	r_ApparentPower					: REAL;
	r_ActivePower					: REAL;
	r_ReactivePower					: REAL;
	r_ACVoltageD7					: REAL;
	r_VoltageDroop					: REAL;
	r_ACVoltageSupply				: REAL;
	r_FrequencyD7					: REAL;
	r_FrequencyDroop				: REAL;
	r_FrequencySupply				: REAL;
	r_CurrentUnbalance				: REAL;
	r_DCPower						: REAL;
	r_DCVoltage						: REAL;
	r_DCCurrent						: REAL;
	r_ACCurrent						: REAL;
	r_ActiveCurrent					: REAL;
	r_ReactiveCurrent				: REAL;
	r_LoadPercent					: REAL; //%
	r_D7SyncError					: REAL;
	r_Pmin							: REAL;
	r_Pmax							: REAL;
	r_QMax							: REAL;
	r_Qmin							: REAL;
	r_Pset							: REAL;
	r_Qset							: REAL;
	r_ACcurrentLimit				: REAL; 
	r_OverCurrentValue				: REAL; // overcurrent ratio 0 .. 1.25 x rated current
	r_ModulationIndex				: REAL;
	
	r_TemperatureInverter			: REAL;
	r_TemperatureGridChoke			: ARRAY [1..3] OF REAL;
	r_TemperatureCMChoke			: ARRAY [1..4] OF REAL;
	r_TemperatureMax				: REAL;
	AddTemperatures					: ST_Inverter_additionalTemperatures;
	w_TemperatureFaultWord			: WORD;
	w_OperationHours				: WORD;
	
	e_PowerMode						: ePowerModes;
	e_InverterMode					: eInverterModes;
	e_Status						: eStatusPowermodule;
	e_ThrottlingStatus					: ePowerModuleThrottlingState;		
	ui_InverterCommStatus			: UINT;
	ui_BuscouplerCommStatus			: UINT;
	
	b_MccbTripOK					: BOOL;
	b_MccbUvr24VdcOK				: BOOL;
	b_MccbFb						: BOOL;
	b_FanFb							: BOOL;
	b_DCcontactorFb					: BOOL;
	b_PrechargeContactor			: BOOL;
	b_LimiterActive					: BOOL;
	
	
	StatusWord						: ST_Inverter_StatusWord;
	UgridStatusWord					: ST_Inverter_UgridStatusWord;
	GridcodeStatusWord				: ST_Inverter_LineState;
	Events							: ST_Powermodule_Events;
	controldata						: ST_Inverter_write;
	
END_STRUCT
END_TYPE

// ---- POUs/Objects/PowerStack/_Structs/ST_PowerModule_set.TcDUT
TYPE ST_PowerModule_set :
STRUCT
	//commands
	r_ActivePower					: REAL;
	r_ReactivePower					: REAL;
	r_NomFrequency					: REAL;
	r_NomVoltage					: REAL;
	r_FrequencyDroop				: REAL;
	r_VoltageDroop					: REAL;
	r_Pmax							: REAL;
	r_Pmin							: REAL;
	r_ACcurrentLimit				: REAL;
	i_PowerChangeRate				: INT; // % nominal power / s
	r_overcurrentFactor				: REAL;
	r_DroopMinimum					: REAL := 0.1;
	r_DroopIslandMode				: REAL := 0.1;
	r_DroopMaximum					: REAL := 10; //%
	
	//WRITE DATA Buscoupler
	b_FanContactor					: BOOL;
	b_D7SyncRequest					: BOOL;
	b_QuickstopInactive				: BOOL;
	b_gridcodeEnable				: BOOL;
	b_ExtgridCodeTrip				: BOOL;
END_STRUCT
END_TYPE

// ---- POUs/Objects/PowerStack/_Structs/ST_Powerstack_Calibration.TcDUT
TYPE ST_Powerstack_Calibration:
STRUCT
	Master				: ST_PowerModule_calibration;
	Slave				: ST_PowerModule_calibration;
END_STRUCT
END_TYPE

// ---- POUs/Objects/PowerStack/_Structs/ST_PowerStack_get.TcDUT
TYPE ST_PowerStack_get :
STRUCT
	// ENUMS
	e_State							: eStatusPowerStack;
	e_PowerState					: ePowerstate;
	e_InverterMode					: eInverterModes;			//0=AFE, Micro, Island, transition
	e_PowerMode						: ePowerModes;				//0=IsoChronous, 1= Droop
	e_ThrottlingStatus				: ePowerModuleThrottlingState;
	
	//POWER DATA (REALS)
	r_VoltageDroop					: REAL;				
	r_FrequencyDroop				: REAL;
	r_ACVoltageD7					: REAL; 
	r_FrequencyD7					: REAL; 
	r_ActivePower					: REAL;
	r_ReactivePower					: REAL;
	r_Pmin							: REAL;
	r_Pmax							: REAL; 
	r_QMax							: REAL;
	r_QMin							: REAL;	
	r_Smax							: REAL;
	r_ACcurrentLimit				: REAL;
	r_ACcurrentLimitMax				: REAL;
	r_PowerChangeRate				: REAL;
	r_ApparentPower					: REAL;
	r_CosPhi						: REAL;
	r_AcCurrent						: REAL;
	r_DCPower						: REAL;
	r_DCVoltage						: REAL;
	r_DCcurrent						: REAL;
	r_ACVoltageSupply				: REAL;
	r_FrequencySupply				: REAL;
	r_LoadPercent					: REAL; //%
	r_RatedCurrent					: REAL;
	r_RatedPower					: REAL;
	r_OvercurrentValueAct			: REAL; //actual overcurrent value
	r_OvercurrentValueMax			: REAL; //max overcurrent value
	r_ThrottlingValueAct			: REAL; // %percentage , inverse of overcurrent with 100%
	
	//Booleans
	b_GridTied						: BOOL;
	b_GridCodeCheckActive			: BOOL;
	b_GridCodeOK					: BOOL := TRUE;
	b_GridACdetected				: BOOL;
	b_InverterGridFormingMode		: BOOL;
	b_ACDetected					: BOOL;
	b_DCDetected					: BOOL;
	b_InverterRunning				: BOOL;
	b_StartedState					: BOOL;
	b_ControlEnabled				: BOOL;
	b_EcomodeAvailable				: BOOL;
	b_StartEnabled					: BOOL;				

	//Temperatures
	r_MaxTemperature				: REAL;
	
	//timers
	t_ShiftHoldTimeRemaining		: TIME;
	t_GridCodeReconnectTime			: TIME;
	//structs
	Events							: ST_PowerStack_Events;
	
	//Sublevel data
	PowermoduleMaster				: REFERENCE TO ST_PowerModule_get();
	PowermoduleSlave				: REFERENCE TO ST_PowerModule_get();
	Netcontactor					: REFERENCE TO ST_Netcontactor_get();
	
END_STRUCT
END_TYPE

// ---- POUs/Objects/PowerStack/_Structs/ST_Powerstack_LOMParams.TcDUT
TYPE ST_Powerstack_LOMParams :
STRUCT
	ForceSlowDetection	: BOOL := FALSE;
	FreqFilterLength	: UINT := 5; // samples 
	DetectionTimeFast_ms: UINT := 50; // milliseconds
	DetectionTimeSlow_ms: UINT := 1000; // milliseconds
	RoCofLimit			: REAL := 0.5; // Hz/s
	PowerPulseSize		: REAL := 0.5; // %, of rated power during ugrid to enable LOM detection.
	EnablePowerPulse	: BOOL := TRUE;
END_STRUCT
END_TYPE

// ---- POUs/Objects/PowerStack/_Structs/ST_PowerStack_params.TcDUT
TYPE ST_PowerStack_params :
STRUCT
	b_SoftStartEnable		: BOOL := TRUE;
	b_StandbyEnable			: BOOL := TRUE;
	b_GridcodesEnabled		: BOOL := TRUE;
	r_DroopMinimum			: REAL := 0.0;
	r_DroopIslandMode		: REAL := 0.1;
	r_DroopMaximum			: REAL := 10; //%
	r_ReactiveOffset		: REAL := 0;
	ui_DeratingStack		: UINT := 5; // %
	ui_DeratingLimCooling	: UINT := 80; // %
	i_MaxPowerChangeRate	: INT := 500; // %/s
	ui_OvercurrentRating	: UINT := 150; // %
	i_ChargeOnlyIdlePower	: INT := -3;
	r_ActiveSetpointGain	: REAL := 1; 
	r_ReactiveSetpointGain  : REAL := 1;
	
	//AC drive limits
	r_FreqLowLimit			: REAL := 48;
	r_FreqHighLimit			: REAL := 52; 
	ui_FreqLimitTripDelay	: UINT := 2000; // milliseconds
	FreqVoltageShift		: st_powerstack_ShiftingParams;
	
	PowermoduleMaster		: ST_PowerModule_params;
	PowermoduleSlave		: ST_PowerModule_params;
	LOM						: ST_Powerstack_LOMParams;
END_STRUCT
END_TYPE

// ---- POUs/Objects/PowerStack/_Structs/ST_PowerStack_Set.TcDUT
TYPE ST_PowerStack_Set :
STRUCT
	//WRITE
	b_NetcontactorHoldClose			: BOOL; // used when input breaker or external PSB breaker must be controlled instead of netcontactor.
	b_ExtGridConnected				: BOOL;
	b_DisableShifting				: BOOL;
	b_slowLom						: BOOL;
	b_automaticswitching			: BOOL;
	b_GridCodeEnable				: BOOL := TRUE;
	e_InverterMode					: eInverterModes;			//0=AFE, 1= ugrid, 2, island
	e_PowerMode						: ePowerModes;				//
	e_NetconClosingRequest			: eNetcontMode;
	e_PowerLimitingMode				: ePLM;
	r_VoltageDroop					: REAL;				
	r_FrequencyDroop				: REAL;
	r_NominalOutputVoltage			: REAL := 400; //R/W
	r_NominalOutputFrequency		: REAL := 50; //R/W
	r_ActivePower					: REAL; //R/W
	r_ReactivePower					: REAL; //R/W
	
	//limits
	r_Pmax							: REAL;
	r_Pmin							: REAL;
	r_ACcurrentLimit				: REAL;
	
END_STRUCT
END_TYPE

// ---- POUs/Objects/ProtectionSystems/FireDetection/_Enums/eCOAlarmStatus.TcDUT
{attribute 'qualified_only'}
{attribute 'strict'}
{attribute 'tostring'}
TYPE eCOAlarmStatus :
(
	Error			:= 0,
	Normal 			:= 1,
	WarningLevel1 	:= 2,
	WarningLevel2 	:= 3,
	Alarm 			:= 4
);
END_TYPE

// ---- POUs/Objects/ProtectionSystems/FireDetection/_Enums/eSmokeDetectAlarmStatus.TcDUT
{attribute 'qualified_only'}
{attribute 'strict'}
{attribute 'tostring'}
TYPE eSmokeDetectAlarmStatus :
(
	Error := 0,
	Normal := 1,
	Alarm := 2
);
END_TYPE

// ---- POUs/Objects/ProtectionSystems/FireDetection/_Structs/ST_CODetectors.TcDUT
TYPE ST_CODetectors :
STRUCT
	State 			: 	eCOAlarmStatus;
	b_CoValuesOK	: 	BOOL;
	Value 			:  	ARRAY[0..3] OF REAL;	//-1 if inoperative. [0]=mean [1]=CO1 [2]=CO2 [3]=max
END_STRUCT
END_TYPE

// ---- POUs/Objects/ProtectionSystems/FireDetection/_Structs/ST_FireDetection_get.TcDUT
TYPE ST_FireDetection_get :
STRUCT
	b_FireAlarm		: 	BOOL;
	SmokeDetectors 	:	ST_SmokeDetectors;
	CODetectors		:	ST_CODetectors;
	Events			:	ST_FireSystem_Events;
END_STRUCT
END_TYPE

// ---- POUs/Objects/ProtectionSystems/FireDetection/_Structs/st_Firedetection_params.TcDUT
TYPE st_Firedetection_params :
STRUCT
	r_COwarningLevel_1				: REAL := 10;
	r_COwarningLevel_2				: REAL := 20;
	r_COalarmLevel					: REAL := 120;
	r_COrange						: REAL := 500;
END_STRUCT
END_TYPE

// ---- POUs/Objects/ProtectionSystems/FireDetection/_Structs/ST_FireDetection_set.TcDUT
TYPE ST_FireDetection_set :
STRUCT
	SilenceSounder	:	BOOL; //only disables currently activated alarm.
	TestSounder		:	BOOL;
END_STRUCT
END_TYPE

// ---- POUs/Objects/ProtectionSystems/FireDetection/_Structs/ST_FireSystem_Events.TcDUT
TYPE ST_FireSystem_Events :
STRUCT
	CODetFault		:	BOOL;
	CODetWarning1	:	BOOL;
	CODetWarning2	: 	BOOL;
	CODetAlarm		:	BOOL;
	SmokeDetFault	:	BOOL;
	SmokeDetAlarm	:	BOOL;
	AlarmMuted		:	BOOL;
END_STRUCT
END_TYPE

// ---- POUs/Objects/ProtectionSystems/FireDetection/_Structs/ST_SmokeDetectors.TcDUT
TYPE ST_SmokeDetectors :
STRUCT
	State : eSmokeDetectAlarmStatus;
END_STRUCT
END_TYPE

// ---- POUs/Objects/ProtectionSystems/FireDetection/_Structs/ST_SmokeDetIO.TcDUT
TYPE ST_SmokeDetIO :
STRUCT
	Signal_OK 	: BOOL;
	Power_OK 	: BOOL;
END_STRUCT
END_TYPE

// ---- POUs/Objects/ProtectionSystems/InsulationMonitoring/_Structs/ST_InsulationMonitor_get.TcDUT
TYPE ST_InsulationMonitor_get :
STRUCT
	b_Enabled							: BOOL;	
	b_PENlinkDetected					: BOOL;
	b_Warning							: BOOL;
	e_EarthingSystemDetected			: eEarthingSystems;
	b_PENlinkOperatedFault				: BOOL;
	b_EarthingSystemMismatch			: BOOL;
	b_NoEarthingSystemSet				: BOOL;
END_STRUCT
END_TYPE

// ---- POUs/Objects/ProtectionSystems/InsulationMonitoring/_Structs/ST_InsulationMonitor_params.TcDUT
TYPE ST_InsulationMonitor_params :
STRUCT
	i_EarthSystemDetectionDelay		:INT := 60; // Seconds
END_STRUCT
END_TYPE

// ---- POUs/Objects/ProtectionSystems/InsulationMonitoring/_Structs/St_InsulationMonitor_PassThrough.TcDUT
TYPE St_InsulationMonitor_PassThrough :
STRUCT
	b_NetContFB				: BOOL;
	b_MccbfbMaster			: BOOL;
	b_MccbfbSlave			: BOOL;
	b_ACdetected			: BOOL;
	b_PENlinkFB				: BOOL;	
END_STRUCT
END_TYPE

// ---- POUs/Objects/ProtectionSystems/InsulationMonitoring/_Structs/ST_InsulationMonitor_set.TcDUT
TYPE ST_InsulationMonitor_set :
STRUCT
	b_enable			: BOOL;
 	e_EarthingSystem	: eEarthingSystems := eEarthingSystems.TN;
END_STRUCT
END_TYPE

// ---- POUs/Objects/ProtectionSystems/OvercurrentProtection/_Structs/ST_OvercurrentProtection_Events.TcDUT
TYPE ST_OvercurrentProtection_Events :
STRUCT
	Input	:ARRAY [1..2] OF ARRAY [1..4] OF FB_Overcurrentdetect(); //FB_UpperLimitAndTimeExceeded();
	Output	:ARRAY [1..3] OF ARRAY [1..4] OF FB_Overcurrentdetect();
END_STRUCT
END_TYPE

// ---- POUs/Objects/ProtectionSystems/OvercurrentProtection/_Structs/ST_OvercurrentProtection_get.TcDUT
TYPE ST_OvercurrentProtection_get :
STRUCT
	//Overcurrent Powerlocks
	r_TotalOutputCurrentLimit			: REAL := 0;
	r_TotalInputCurrentLimit			: REAL := 0;
	b_OutputWarning						: BOOL;
	b_InputWarning						: BOOL;
	b_OutputAlarm						: BOOL;
	b_InputAlarm						: BOOL;
	r_PeakCurrent						: REAL;
	t_PeakCurrentDuration				: TIME;
	s_locationPeak						: STRING;
	
	Events								: ST_OvercurrentProtection_events;
END_STRUCT
END_TYPE

// ---- POUs/Objects/ProtectionSystems/OvercurrentProtection/_Structs/ST_OvercurrentProtection_InternalLinking.TcDUT
TYPE ST_OvercurrentProtection_InternalLinking :
STRUCT
	a_r_CurrentInput			: ARRAY [1..2] OF ARRAY[1..4] OF REAL; //first array of powerlockset, second of powerlock
	a_r_CurrentOutput			: ARRAY [1..3] OF ARRAY[1..4] OF REAL;
	b_InputSectionAvailable 	: BOOL;
	b_thirdOutputAvailable 		: BOOL;
END_STRUCT
END_TYPE

// ---- POUs/Objects/ProtectionSystems/OvercurrentProtection/_Structs/ST_OvercurrentProtection_Params.TcDUT
TYPE ST_OvercurrentProtection_Params :
STRUCT
	ui_OCPtripTime		: UINT := 900; //Seconds
	ui_Ik				: UINT := 16; // Short circuit capacity of component to be protected [Ik/s]
	ui_Irated			: UINT := 400; // rated current 
	ui_gain				: UINT := 10; //gain for tuning calculated remaining time during overcurrent.
	OutputNormalShutdownDelay : TIME := T#5S;
END_STRUCT
END_TYPE

// ---- POUs/Objects/ProtectionSystems/OvercurrentProtection/_Structs/ST_OvercurrentProtection_set.TcDUT
TYPE ST_OvercurrentProtection_set :
STRUCT
	ui_PowerlockInputCurrentLimit			: ARRAY [1..2] OF UINT := [400,400];
	ui_PowerlockOutputCurrentLimit			: ARRAY [1..3] OF UINT := [400,400,400];
END_STRUCT
END_TYPE

// ---- POUs/Objects/ProtectionSystems/ResidualCurrentMonitoring/_Structs/ST_ResidualCurrentMonitor_get.TcDUT
TYPE ST_ResidualCurrentMonitor_get :
STRUCT
	b_prewarning			: BOOL;
END_STRUCT
END_TYPE

// ---- POUs/Objects/ProtectionSystems/SurgeProtection/_Structs/ST_Surgeprotection_get.TcDUT
TYPE ST_Surgeprotection_get :
STRUCT
	b_Type12_OK				: BOOL;
	b_Type3_OK				: BOOL;			
END_STRUCT
END_TYPE

// ---- POUs/Objects/ProtectionSystems/_Struct/ST_ProtectionSystems_get.TcDUT
TYPE ST_ProtectionSystems_get :
STRUCT
	//Fire Detection System
	FireDetection						: ST_Firedetection_get;
	
	//InsulationMonitor
	Insulation							: ST_InsulationMonitor_get;
	
	//MRCDB
	MRCDB								: ST_ResidualCurrentMonitor_get;
	
	//Surge protection
	Surge								: ST_SurgeProtection_get;
	
	//Overcurrent protection
	OvercurrentProtection				: ST_OverCurrentProtection_Get;
	
END_STRUCT
END_TYPE

// ---- POUs/Objects/ProtectionSystems/_Struct/ST_ProtectionSystems_Params.TcDUT
TYPE ST_ProtectionSystems_Params :
STRUCT
	InsulationMonitor				: ST_InsulationMonitor_params;
	firedetection					: ST_Firedetection_params;
	OCP								: ST_Overcurrentprotection_params;
END_STRUCT
END_TYPE

// ---- POUs/Objects/ProtectionSystems/_Struct/ST_ProtectionSystems_set.TcDUT
TYPE ST_ProtectionSystems_set :
STRUCT
	//Fire Detection System
	FireDetection						: ST_Firedetection_set;
	
	//InsulationMonitor
	Insulation							: ST_InsulationMonitor_set;
	
	//OCP
	OvercurrentProtection				: ST_OvercurrentProtection_set;
END_STRUCT
END_TYPE

// ---- POUs/Objects/PeakshaveBox/DUTs/eWago750495_ACDataID_1.TcDUT
{attribute 'qualified_only'}
{attribute 'strict'}
{attribute 'to_String'}
TYPE eWago750495_ACDataID_1 :
(
	//only RMS and peak values are declared
	//Voltages
	VoltageL1N_RMS			:= 4,
	VoltageL2N_RMS 			:= 5,
	VoltageL3N_RMS			:= 6,
	VoltageL1L2_RMS			:= 31,
	VoltageL2L3_RMS 		:= 32,
	VoltageL3L1_RMS			:= 33,
	VoltageL1N_Peak 		:= 91,
	VoltageL2N_Peak 		:= 92,
	VoltageL3N_Peak 		:= 93,
	
	//Currents
	CurrentL1_RMS			:= 1,
	CurrentL2_RMS			:= 2,
	CurrentL3_RMS			:= 3,
	CurrentN_RMS			:= 97,
	CurrentL1_Peak			:= 94,
	CurrentL2_Peak			:= 95,
	CurrentL3_Peak			:= 96,
	                           
	//Power                    
	ActivePowerL1			:= 07,
	ActivePowerL2			:= 08,
	ActivePowerL3			:= 09,
	ReactivePowerL1			:= 10,
	ReactivePowerL2			:= 11,
	ReactivePowerL3			:= 12,
	ApparentPowerL1			:= 13,
	ApparentPowerL2			:= 14,
	ApparentPowerL3			:= 15,
	
	//Energy
	ActiveEnergyTotal			:= 73,
	ActiveEnergyImport			:= 74,
	ActiveEnergyExport			:= 75,
	ReactiveEnergyTotal			:= 85,
	ReactiveEnergyInductive		:= 86,
	AReactiveEnergyCapacitive	:= 87,
	
	//Frequency
	FrequencyL1				:= 16,
	FrequencyL2				:= 17,
	FrequencyL3				:= 18,
	                           
	//Phase Angle              
	PhaseAngleL1			:= 19,
	PhaseAngleL2			:= 20,
	PhaseAngleL3			:= 21,
	
	//PowerFactor
	PowerFactorL1			:= 25,
	PowerFactorL2			:= 26,
	PowerFactorL3			:= 27
) USINT;
END_TYPE

// ---- POUs/Objects/PeakshaveBox/DUTs/eWago750495_HarmonicsDataID_1.TcDUT
{attribute 'qualified_only'}
{attribute 'strict'}
{attribute 'to_String'}
TYPE eWago750495_HarmonicsDataID_1 :
(
	Current_RMS 		:= 001,
	Voltage_RMS 		:= 002,
	CurrentTHD			:= 003,
	VoltageTHD			:= 004
	
	//harmonics not declared for now
);
END_TYPE

// ---- POUs/Objects/PeakshaveBox/DUTs/eWago750495_MeasureGroupID_1.TcDUT
{attribute 'qualified_only'}
{attribute 'strict'}
{attribute 'to_String'}
TYPE eWago750495_MeasureGroupID_1 :
(
	ac := 10,
	harmonicsL1 := 20,
	harmonicsL2 := 21,
	harmonicsL3	:= 22
) USINT;
END_TYPE

// ---- POUs/Objects/PeakshaveBox/DUTs/eWago750495_StatDataID_1.TcDUT
{attribute 'qualified_only'}
{attribute 'strict'}
TYPE eWago750495_StatDataID_1 :
(
	Phase1 := 0,
	Phase2 := 1,
	Phase3 := 2,
	IOmodule:= 3
)USINT;
END_TYPE

// ---- POUs/Objects/PeakshaveBox/DUTs/ST_Wago750495_Data_1.TcDUT
TYPE ST_Wago750495_Data_1 :
STRUCT
	//Voltages
	r_VoltageL1N_RMS				: REAL;
	r_VoltageL2N_RMS 				: REAL;
	r_VoltageL3N_RMS				: REAL;
	r_VoltageL1L2_RMS				: REAL;
	r_VoltageL2L3_RMS 				: REAL;
	r_VoltageL3L1_RMS				: REAL;
	r_VoltageL1N_Peak 				: REAL;
	r_VoltageL2N_Peak 				: REAL;
	r_VoltageL3N_Peak 				: REAL;
	                            	      
	//Currents                  	      
	r_CurrentL1_RMS					: REAL;
	r_CurrentL2_RMS					: REAL;
	r_CurrentL3_RMS					: REAL;
	r_CurrentN_RMS					: REAL;
	r_CurrentL1_Peak				: REAL;
	r_CurrentL2_Peak				: REAL;
	r_CurrentL3_Peak				: REAL;
	                            	      
	//Power                     	      
	r_ActivePowerL1					: REAL;
	r_ActivePowerL2					: REAL;
	r_ActivePowerL3					: REAL;
	r_ReactivePowerL1				: REAL;
	r_ReactivePowerL2				: REAL;
	r_ReactivePowerL3				: REAL;
	r_ApparentPowerL1				: REAL;
	r_ApparentPowerL2				: REAL;
	r_ApparentPowerL3				: REAL;
	
	//Energy
	r_ActiveEnergyTotal				: REAL;
	r_ActiveEnergyImport			: REAL;
	r_ActiveEnergyExport			: REAL;
	r_ReactiveEnergyTotal			: REAL;
	r_ReactiveEnergyInductive		: REAL;
	r_AReactiveEnergyCapacitive		: REAL;
	
	//Frequency
	r_FrequencyL1					: REAL;
	r_FrequencyL2					: REAL;
	r_FrequencyL3					: REAL;
	                        		      
	//Phase Angle           		      
	r_PhaseAngleL1					: REAL;
	r_PhaseAngleL2					: REAL;
	r_PhaseAngleL3					: REAL;
	                        		      
	//PowerFactor           		      
	r_PowerFactorL1					: REAL;
	r_PowerFactorL2					: REAL;
	r_PowerFactorL3					: REAL;
	
	
END_STRUCT
END_TYPE

// ---- POUs/Objects/PeakshaveBox/DUTs/ST_Wago750495_ExtStatusWord_1.TcDUT
TYPE ST_Wago750495_ExtStatusWord_1 :
STRUCT
	b_IncreasedMeasErr			: BOOL; //Stat 1 query L1,L2,L3:: increase measurement error of selected phase
	b_CurrentClipping			: BOOL; //Stat 2 query L1,L2,L3:: current out of measurable range of selected phase
	b_VoltageClipping			: BOOL; //Stat 3 query L1,L2,L3:: voltage out of measurable range of selected phase
	b_NoZeroCrossings			: BOOL; //Stat 4 query L1,L2,L3:: Zero Crossings missing of selected phase
	b_OverCurrent				: BOOL; //Stat 5 query L1,L2,L3:: Overcurrent of selected phase
	b_OverVoltage				: BOOL; //Stat 6- query L1,L2,L3: OverVoltage of selected phase.
	b_RotaryField				: BOOL; //Stat 6- query IO: 0:Clockwise, 1: counterclockwise
	b_UnderVoltage				: BOOL; //Stat 7- query L1,L2,L3: UnderVoltage of selected phase

END_STRUCT
END_TYPE

// ---- POUs/Objects/PeakshaveBox/DUTs/ST_Wago750495_Read_1.TcDUT
TYPE ST_Wago750495_Read_1 :
STRUCT
	StatusWord				: ST_Wago750495_StatusWord;
	ExtStatusWord			: ST_Wago750495_ExtStatusWord;
	Data					: ST_Wago750495_Data;
END_STRUCT
END_TYPE

// ---- POUs/Objects/PeakshaveBox/DUTs/ST_Wago750495_StatusWord_1.TcDUT
TYPE ST_Wago750495_StatusWord_1 :
STRUCT
	b_ComFb						: BOOL; // 0: process Data, 1: Register Data
	b_Error						: BOOL; // 0: OK, 1: Error
	b_Error_IO					: BOOL; // 0: OK, 1: Error
	b_Error_L3					: BOOL; // 0: OK, 1: Error
	b_Error_L2					: BOOL; // 0: OK, 1: Error
	b_Error_L1					: BOOL; // 0: OK, 1: Error
	e_StatIDfb					: eWago750495_StatDataID;
	b_Warning					: BOOL; // 0: OK, 1: Transient reaction measured value collection active
	b_Cal						: BOOL; // 0: Measurement Mode, 1: Calibration Mode
	b_Over_1					: BOOL; // 0: OK, 1: Out Of Range
	b_Over_2					: BOOL; // 0: OK, 1: Out Of Range
	b_Over_3					: BOOL; // 0: OK, 1: Out Of Range
	b_Over_4					: BOOL; // 0: OK, 1: Out Of Range
	e_GroupID					: eWago750495_MeasureGroupID;

END_STRUCT
END_TYPE

// ---- POUs/Objects/PeakshaveBox/DUTs/ST_Wago750495_Write_1.TcDUT
TYPE ST_Wago750495_Write_1 :
STRUCT
	b_EnableRegisterComm		: BOOL;
	e_statusQuery				: eWago750495_StatDataID; //0: status L1, 1: status L2, 2: Status L3, 3: Status IO Module			
END_STRUCT
END_TYPE

// ---- POUs/Objects/PeakshaveBox/ST_PeakShaveBox_Get.TcDUT
TYPE ST_PeakShaveBox_Get :
STRUCT
	PSBmode				: ePSBMode;
	Powermonitor 		: st_MeasurementVoltageData;
	PowerStatus			: st_PowerMeasurement_status;
	r_MaxCTCurrent		: REAL:= 4000;
	b_buscouplerReady	: BOOL;
	b_active			: BOOL;
	b_dataOK			: BOOL;
	b_ContactorFb		: BOOL;
	b_SyncFb			: BOOL;
	b_SettingsChangePending	:	BOOL;
END_STRUCT
END_TYPE

// ---- POUs/Objects/WearLogging/eEntryType.TcDUT
{attribute 'qualified_only'}
{attribute 'strict'}
TYPE eEntryType :
(
	IntegerValue		:=	0,
	FloatValue			:=	1,
	StringValue			:=	2
);
END_TYPE

// ---- POUs/Objects/WearLogging/eLogItemGroupID.TcDUT
{attribute 'qualified_only'}
{attribute 'to_string'}
TYPE eLogItemGroupID :
(	
	//None					:= 	0,
	General					:=	1,
	ACSwitchgear			:=	2,
	CoolingSystem			:=	3,
	BMS						:=	4,
	PowerStack				:=	5,
	Enclosure				:=	6,
	InternalPowerSupply		:=	7,
	Safety					:=	8,
	ZPT						:=  9
) WORD := General;
END_TYPE

// ---- POUs/Objects/WearLogging/eLogTypes.TcDUT
{attribute 'qualified_only'}
{attribute 'strict'}
TYPE eLogTypes :
(
	TrackCycles := 0,
	TrackOnTime	:= 1,
	WriteValue := 2,
	KeepHighestValue := 3,
	KeepLowestValue	:= 4
);
END_TYPE

// ---- POUs/Objects/WearLogging/LogState.TcDUT
{attribute 'qualified_only'}
{attribute 'strict'}
TYPE LogState :
(
	Init 			:= 0,
	Loading_file 	:= 1,
	Idle			:= 3,
	SavingLogData	:= 4,
	
	FileNotFound	:= 99
);
END_TYPE

// ---- POUs/Safety/ST_Safety_ContactorEDM.TcDUT
TYPE ST_Safety_ContactorEDM :
STRUCT
	b_MccbMasterEDM						: BOOL;
	b_MccbSlaveEDM						: BOOL;
	b_NetcontactorEDM					: BOOL;
END_STRUCT
END_TYPE

// ---- POUs/Safety/ST_Safety_get.TcDUT
TYPE ST_Safety_get :
STRUCT
	b_SafetyOK					: BOOL;
	b_EstopChannelAOK			: BOOL;		
	b_EstopChannelBOK			: BOOL;		
	b_InsulationMonitorOK		: BOOL;	
	b_MRCDBOK					: BOOL;	
	b_InverterDoorOK            : BOOL;
	b_ZptOK				        : BOOL;
END_STRUCT
END_TYPE

// ---- POUs/Safety/ST_Safety_ToSafetyPrg.TcDUT
TYPE ST_Safety_ToSafetyPrg :
STRUCT
	b_ErrorReset						: BOOL;
	b_SafetyPrgReset					: BOOL;
	b_EmergencyStopSoftwareOK			: BOOL;
	b_SafetyRunStop						: BOOL := TRUE;
	contactors							: ST_Safety_ContactorEDM;
END_STRUCT
END_TYPE

// ---- POUs/System/GenGridControl/_enums/eBreakerOperationMode.TcDUT
{attribute 'qualified_only'}
{attribute 'strict'}
{attribute 'to_string'}

TYPE eBreakerOperationMode :
(
	none 				:= 0,
	GridFeedthrough		:= 1,
	ExtGrid				:= 2,
	GenDroop			:= 3,
	GenIso				:= 4,
	GenFix				:= 5
);
END_TYPE

// ---- POUs/System/GenGridControl/_enums/eGenIsoInverterMode.TcDUT
{attribute 'qualified_only'}

TYPE eGenIsoInverterMode:
(
	AFE := 0,
	ISO_CUSTOMDROOP := 1,
	ISO_SLOWDROOP:= 2
);
END_TYPE

// ---- POUs/System/GenGridControl/_enums/eGensetStartStop.TcDUT
{attribute 'qualified_only'}
{attribute 'strict'}
TYPE eGensetStartStop :
(
	Auto := 0,
	Stop := 1,
	Start := 2
);
END_TYPE

// ---- POUs/System/GenGridControl/_enums/eGensetMode.TcDUT
{attribute 'qualified_only'}
{attribute 'strict'}
{attribute 'to_string'}
TYPE eGensetMode :
(
	Isochronous := 0,
	Droop := 1,
	FixedPower := 2
);
END_TYPE

// ---- POUs/System/GenGridControl/_enums/ePowerControlMode.TcDUT
{attribute 'qualified_only'}
{attribute 'strict'}
{attribute 'to_string'}
TYPE ePowerControlMode :
(
	None 						:= 0,
	PeakshaveExt 				:= 1,
	PeakshaveInputGrid 			:= 2,
	PeakshaveInputGen 			:= 3
);
END_TYPE

// ---- POUs/System/GenGridControl/_enums/eGenGridState.TcDUT
{attribute 'qualified_only'}
{attribute 'strict'}
{attribute 'to_string'}

TYPE eGenGridState :
(
	Init := 0,
	Idle := 1, 
	Waiting_Trigger := 2,
	Starting := 3,
	Running := 4,
	Stopping := 5,
	Warmup := 6,
	Cooldown := 7,
	Synchronization := 8,
	Waiting_Mode_Reconnect := 9,
	Gridcode_Release_Check := 10,
	Waiting_For_AC := 11
);
END_TYPE

// ---- POUs/System/GenGridControl/_enums/eRunCondition.TcDUT
{attribute 'qualified_only'}
{attribute 'strict'}
TYPE eRunCondition :
(
	None := 0,
	SoC := 1,
	DischargeOverload := 2,
	BattFull := 3,
	ChargeOverload := 4,
	ManuallyStarted := 5,
	ManuallyStopped := 6
);
END_TYPE

// ---- POUs/System/GenGridControl/_structs/ST_ContactorControl_params.TcDUT
TYPE ST_ContactorControl_params :
STRUCT
	ui_VoltageDevSyncOK			: UINT := 4;
	ui_DeloadCurrentRelease		: UINT := 20;
	ui_DeloadTimeOut			: UINT := 60; //s
	VoltagePID					: st_Powercontrol_PIDparams := (Enable:= TRUE, kp:=0.5, Tv:=0, Tn:=1000, Td:=0, Outerwindow:= 0, Innerwindow := 0, OutputDeadband := 0, InputDeadband := 0.5);
END_STRUCT
END_TYPE

// ---- POUs/System/GenGridControl/_structs/ST_GenGridController_Events.TcDUT
TYPE ST_GenGridController_Events :
STRUCT
	b_InvalidGensetParameters 		: BOOL;
	b_RotationFieldFault			: BOOL;
	b_CurrentLimitDisconnect		: BOOL;
	b_CurrentLimitTrip				: BOOL;
	b_EmstopDisconnect				: BOOL;
	b_ShutdownDisconnect			: BOOL;
	b_OverloadTrip  				: BOOL;
	b_OverFreqTrip					: BOOL;
	b_UnderFreqTrip					: BOOL;
	b_OverVoltTrip					: BOOL;
	b_UnderVoltTrip					: BOOL;
	b_ShutdownTimeOut				: BOOL;
	b_SynchronisationFault			: BOOL;
	b_StartupFault					: BOOL;
	b_WarmupFault					: BOOL;
	b_GenDownTrip					: BOOL;
	b_GridLostTrip					: BOOL;
	b_TransToGenIsoInhibit			: BOOL;
	b_TransToGenDroopInhibit		: BOOL;
	b_TransToGenFixInhibit			: BOOL;
	b_TransFromInputGridAckRQ		: BOOL;
	b_TransFromInputGenAckRQ		: BOOL;
	b_StartingInhibit				: BOOL;

END_STRUCT
END_TYPE

// ---- POUs/System/GenGridControl/_structs/ST_GenGridController_get.TcDUT
TYPE ST_GenGridController_get :
STRUCT
	b_active			: BOOL;
	b_faultActive		: BOOL;
	b_gensetHot			: BOOL;
	b_gensetStarting	: BOOL;
	b_ModeTransActive	: BOOL;
	b_ModeTransInhibit	: BOOL;
	b_ModeChanged		: BOOL;
	b_ShowModeTrans		: BOOL;
	b_extGensetMode 	: BOOL;
	b_gensetcontrol		: BOOL;
	e_BreakerMode		: eBreakerOperationMode;
	e_PowerControlMode	: ePowerControlMode;
	e_GensetMode		: eGensetMode;
	e_GensetStartStop	: eGensetStartStop;
	e_state				: eGenGridState;
	e_RunCondition		: eRunCondition;
	events				: ST_GengridController_events;
	
END_STRUCT
END_TYPE

// ---- POUs/System/GenGridControl/_structs/ST_GenGridController_Params.TcDUT
TYPE ST_GenGridController_Params :
STRUCT
	r_SocHysteresis				: REAL := 2; //used for auto start/stop
	r_PIDLimitRampDefault		: REAL := 50; // default ramp rate when PID limits are changed
	by_SyncRetries				: BYTE := 5; 
	by_CurrentLimitMargin		: REAL := 20; // Headroom from the current limit where the trip can be detected. 10 = 10A headroom 
	CurrentLimitTripDelay		: TIME := T#5S; // 
	GenIso_InverterMode			: eGenIsoInverterMode := eGenIsoInverterMode.ISO_SLOWDROOP; //inverter mode when operating with genset in iso at input.
	Contactor					: ST_ContactorControl_params;
	Genset						: ST_GengridController_ParamsGenset;
END_STRUCT
END_TYPE

// ---- POUs/System/GenGridControl/_structs/St_GenGridController_ParamsGenset.TcDUT
TYPE St_GenGridController_ParamsGenset :
STRUCT
	OverloadTripDelay	 		: UINT := 3000; //ms
	UnderFrequencyLimit			: REAL := 49;
	UnderfrequencyTripDelay		: UINT := 2000; //ms
	OverFrequencyLimit			: REAL := 51;
	OverfrequencyTripDelay		: UINT := 2000; //ms
	UnderVoltageLimit			: REAL := 360;
	UnderVoltageTripDelay		: UINT := 2000; //ms
	OverVoltageLimit			: REAL := 435;
	OverVoltageTripDelay		: UINT := 2000; //ms
	ShutdownTimeout				: UINT := 180; //s
	GenDownRetries				: BYTE := 3;
	OverloadOffDelay			: TIME := T#10M;
	OverloadOnDelay				: TIME := T#10S;
END_STRUCT
END_TYPE

// ---- POUs/System/GenGridControl/_structs/ST_GenGridController_SyncData.TcDUT
TYPE ST_GenGridController_SyncData :
STRUCT
	b_Sync				: BOOL;
	r_freqSet			: REAL;
	r_VoltSet			: REAL;
END_STRUCT
END_TYPE

// ---- POUs/System/PowerControl/_enums/ePIDmode.TcDUT
{attribute 'qualified_only'}
{attribute 'strict'}
TYPE ePIDmode :
(
	None := 0,
	Q := 1,
	P := 2,
	Both := 3
);
END_TYPE

// ---- POUs/System/PowerControl/_Structs/ST_PowerControl_Events.TcDUT
TYPE ST_PowerControl_Events :
STRUCT
	b_ReactivePIDError			: BOOL;
	b_ActivePIDError			: BOOL;
	b_FreqShiftPIDError			: BOOL;
END_STRUCT
END_TYPE

// ---- POUs/System/PowerControl/_Structs/ST_PowerControl_Get.TcDUT
TYPE ST_PowerControl_Get :
STRUCT
	r_CurrentAct				: REAL; // of the target
	r_Sact						: REAL; // of the target
	r_PAct						: REAL; // of the target
	r_QAct						: REAL; // of the target
	r_PhaseVoltageAct			: REAL; // of the target
	r_PFact						: REAL; // of the target
	
	r_FeedInCurrentLimitActual	: REAL;
	r_SupplyInCurrentLimitActual: REAL;
	
	b_ThrottlingActive			: BOOL;
	ui_ThrottlingType			: UINT; // 0= max watt, 14 = derating
	events						: ST_PowerControl_events;
END_STRUCT
END_TYPE

// ---- POUs/System/PowerControl/_Structs/st_Powercontrol_params.TcDUT
TYPE st_Powercontrol_params :
STRUCT
	//PIDreset				: BOOL; //rising edge
	SocDroop				: ST_PowerControl_SocDroopParams;
	FreqShiftPID			: st_Powercontrol_PIDparams := (Enable:= FALSE, kp:=0.1, Tv:=0, Tn:=1000, Td:=0, Outerwindow:= 0, Innerwindow := 0, OutputDeadband := 0, InputDeadband := 0.05);
	ReactivePID				: st_Powercontrol_PIDparams := (Enable:= TRUE, kp:=5, Tv:=0, Tn:=20, Td:=0, Outerwindow:= 0, Innerwindow := 0, OutputDeadband := 0.5, InputDeadband := 1);
	ActivePID				: st_Powercontrol_PIDparams := (Enable:= TRUE, kp:=5, Tv:=100, Tn:=15, Td:=100, Outerwindow:= 0, Innerwindow := 0, OutputDeadband := 0.5, InputDeadband := 1);
	VoltagePeakshavePID		: st_Powercontrol_PIDparams := (Enable:= TRUE, kp:=1, Tv:=0, 	Tn:=200, Td:=0, Outerwindow:= 0, Innerwindow := 0, OutputDeadband := 0, InputDeadband := 20);
	TransitionRamp			: UINT := 5; // kw & kva per second
	TransitionTime			: UINT := 500; // milliseconds
END_STRUCT
END_TYPE

// ---- POUs/System/PowerControl/_Structs/st_Powercontrol_PIDparams.TcDUT
TYPE st_Powercontrol_PIDparams :
STRUCT
	enable					: BOOL;
	Kp						: REAL;
	Tv						: UINT; //ms
	Tn						: UINT; //ms
	Td						: UINT; //ms
	Outerwindow				: REAL;
	InnerWindow				: REAL;
	OutputDeadband			: REAL;
	InputDeadband			: REAL;
END_STRUCT
END_TYPE

// ---- POUs/System/PowerControl/_Structs/ST_PowerControl_PsTarget_Measurements.TcDUT
TYPE ST_PowerControl_PsTarget_Measurements :
STRUCT
	r_PhaseVoltage					: REAL;
	r_ActivePower					: REAL;
	r_ReactivePower					: REAL;
END_STRUCT
END_TYPE

// ---- POUs/System/PowerControl/_Structs/ST_Powercontrol_set.TcDUT
TYPE ST_Powercontrol_set :
STRUCT
	
END_STRUCT
END_TYPE

// ---- POUs/System/PowerControl/_Structs/ST_PowerControl_SocDroopParams.TcDUT
TYPE ST_PowerControl_SocDroopParams :
STRUCT
	enable				: BOOL := TRUE;
	SocMinDroopStart	: REAL := 20; // at XX%, frequency is shifted linearly down with the actual SOC towards 0%.
	SocMaxDroopStart	: REAL := 80; // at XX%, frequency is shifted linearly up with the actual SOC towards 100%.
END_STRUCT
END_TYPE

// ---- POUs/System/PowerControl/_Structs/ST_PowerControl_Target.TcDUT
TYPE ST_PowerControl_Target :
STRUCT
	PIDmode								: ePIDmode := ePIDmode.Q;
	PeakshaveMode						: BOOL;// for use of genpeakshaving						
	r_PIDRampRate						: REAL;
	r_FeedInCurrentLimit				: REAL; // from battery/loads to peakshave target
	r_SupplyCurrentLimit				: REAL; // from peakshave target to battery/loads
	r_PowerTarget						: REAL;
	b_EnableSocDrooping					: BOOL;
	b_GenIsoPID							: BOOL; // PF = 1 set point enable, Currentlimit is pure active. 
	r_droopMinimum						: REAL;
	Syncdata							: ST_GenGridController_SyncData;
	Measurements						: ST_Powercontrol_PsTarget_Measurements;
END_STRUCT
END_TYPE

// ---- POUs/System/_Structs/ST_SystemTime.TcDUT
TYPE ST_SystemTime :
STRUCT
	AutoSyncToGPS	:	BOOL;
	ManualSync		:	BOOL;
	ManSyncValue	:	DT;
END_STRUCT
END_TYPE

// ---- POUs/System/_Structs/ST_System_Calibration.TcDUT
TYPE ST_System_Calibration :
STRUCT
	Powerstack			: ST_Powerstack_calibration;
END_STRUCT
END_TYPE

// ---- POUs/System/_Structs/ST_System_Events.TcDUT
TYPE ST_System_Events :
STRUCT
	b_RestartRequiredMachineName		: BOOL;
	b_TimeUpdateFailed					: BOOL;
END_STRUCT
END_TYPE

// ---- POUs/System/_Structs/ST_System_params.TcDUT
TYPE ST_System_params :
STRUCT
	//Monitoring & control
	Powercontroller						: ST_Powercontrol_params;
	GenGridController					: ST_GenGridController_params;
	b_VDLReset							: BOOL;
	OutputContactSignal					: eOutputContactSignal := eOutputContactSignal.GenStartStop;
	SystemTime							: ST_SystemTime;
END_STRUCT
END_TYPE

// ---- POUs/System/_Structs/ST_System_Properties.TcDUT
TYPE ST_System_Properties :
STRUCT
	r_RatedActivePower		: 	REAL;
	r_RatedApparentPower	: 	REAL;
	r_RatedCurrent			: 	REAL;
	r_ratedCurrentInput		: 	REAL := 700;
	r_ratedCurrentOutput	: 	REAL;
	r_RatedEnergyCapacity	: 	REAL; // kWh
	r_SelfdischargeRate		: 	REAL := 3; // 3% per month
	s_ProductionDate		: 	STRING;
	s_Weight				: 	STRING;
	s_ManufacturerModel		: 	STRING := 'e-PU10';
	s_ConfigurationCode		: 	STRING;
	s_SerialNumber			: 	STRING;
	by_SWverMajor			:	BYTE;
	by_SWverMinor			:	BYTE;
	by_SWverPatch			:	BYTE;
	by_SWverBuild			:	BYTE;
	s_SWversionNumber		: 	STRING;
	s_Client				: 	STRING;
	r_DischargedEnergy		: 	REAL;
	r_ChargedEnergy			: 	REAL;
END_STRUCT
END_TYPE

// ---- POUs/System/_Structs/ST_System_set.TcDUT
TYPE ST_System_set :
STRUCT
	//structurized variables from function blocks\
	control						: ST_ControlVars;
	powerstack					: ST_Powerstack_Set;
	BMS							: ST_BMS_Set;
	ACSwitchgear				: ST_ACswitchgear_set;
	Peakshavebox				: ST_PeakshaveBox_set;
	Protections					: ST_ProtectionSystems_set;
	Enclosure					: ST_Enclosure_set;
	HartingIO					: ST_HartingIO_set;
	GenComm						: ST_Genset_Set;
	AcDcCharger					: ST_AcDcCharger_set;
	b_TransportMode				: BOOL;
END_STRUCT
END_TYPE

// ---- POUs/System/_Structs/ST_System_get.TcDUT
TYPE ST_System_get :
STRUCT
	b_SMSnumberConfigured		: BOOL;
	b_CustomNameConfigured		: BOOL;
	s_SystemName				: STRING(20);
	b_TransportModePending		: BOOL;
	b_DehumModePending			: BOOL;
	
	
	//Statuss
	e_State						: eSystemState; //0:Idle, 1: Stand-by, 2:Conditioning, 3:Dry-Cycle, 4: Running, 5: Charging only, 6: Discharging only, 7: Stopped 8:Fault, 10: Reset
	e_gridmode					: eGridmode;
	e_UgridPowermode			: eUgridPowermode;
	b_StartAllowed				: BOOL;
	r_CurrentEfficiency			: REAL;
	r_AvgEfficiency				: REAL;
	r_RoundtripEfficiency		: REAL;
	DT_SystemTime				: DT;
	
	PowerController				: ST_PowerControl_get;	
	GenGridController			: ST_GenGridController_get;	
	
	events						: ST_System_events;
END_STRUCT
END_TYPE

// ---- POUs/System/_Structs/ST_System_Monitor.TcDUT
{ attribute 'TcHmiSymbol.ShowRecursively' }

TYPE ST_System_Monitor :
STRUCT
	b_modeSwitchEnable					: BOOL;
	
	safety								: ST_Safety_get;
	system								: ST_System_get;
	powerstack							: REFERENCE TO ST_Powerstack_get;
	powermonitor						: REFERENCE TO ST_PowerMonitor_get;
	AcDcCharger							: REFERENCE TO ST_AcDcCharger_get;
	ACswitchgear						: REFERENCE TO ST_ACSwitchgear_Get;
	neutraltransformer					: REFERENCE TO ST_NeutralTransformer_Get;
	battery								: REFERENCE TO st_BMS_get;
	protections							: REFERENCE TO ST_ProtectionSystems_get;
	peakshavebox						: REFERENCE TO ST_Peakshavebox_get;
	enclosure							: REFERENCE TO ST_Enclosure_get;
	internalpsu							: REFERENCE TO ST_InternalPowersupply_Get;
	DCswitchgear						: REFERENCE TO ST_DCSwitchgear_Get;
	PLC									: REFERENCE TO ST_plcstate_get;
	Cooling								: REFERENCE TO ST_Coolingsystem_get;
	Router								: REFERENCE TO ST_Router_get;
	controlfb							: REFERENCE TO ST_System_Control;
	Generator							: REFERENCE TO ST_Genset_Get;
	HartingIO							: REFERENCE TO ST_HartingIO_Get;
	//Cooling							
END_STRUCT
END_TYPE

// ---- POUs/System/_Structs/ST_System_Control.TcDUT
{ attribute 'allowImplicitAccess'}
TYPE ST_System_Control :
STRUCT
	control				: ST_ControlVars;
	Operation			: ST_OperationVars;
	SoftSettings		: ST_SoftSettings;
	HardSettings		: ST_Hardsettings;
END_STRUCT
END_TYPE

// ---- GVLs/GVL.TcGVL
{attribute 'qualified_only'}
VAR_GLOBAL
	s_SystemTime						: STRING;
	s_SystemDate						: STRING;
	dt_SystemDateTime					: DT;
	b_SystemClockOK						: BOOL;
	b_SystemReady						: BOOL;
	b_initCycle							: BOOL := TRUE;
	b_LEDDemoMode						: BOOL;
	
	
	//error variables
	b_WarningActive						: BOOL;
	b_NormalShutdownActive				: BOOL;
	b_QuickshutdownActive				: BOOL;
	b_EmergencyShutdownActive			: BOOL;	
	

END_VAR

// ---- GVLs/Settings.TcGVL
{attribute 'qualified_only'}
VAR_GLOBAL PERSISTENT
	{ attribute 'TcHmiSymbol.ShowRecursively' }
	Configuration						: ST_System_Config;
	{ attribute 'TcHmiSymbol.ShowRecursively' }
	MachineParams						: ST_System_MachineParams;
	{ attribute 'TcHmiSymbol.ShowRecursively' }
	GridParams							: ST_System_GridCodeParams;
	{ attribute 'TcHmiSymbol.ShowRecursively' }
	Properties							: ST_System_Properties;
	{ attribute 'TcHmiSymbol.ShowRecursively' }
	Calibration							: ST_System_Calibration;
	{ attribute 'TcHmiSymbol.ShowRecursively' }
	Save								: BOOL;
	{ attribute 'TcHmiSymbol.ShowRecursively' }
	Load								: BOOL;
END_VAR

// ---- GVLs/Units.TcGVL
{attribute 'qualified_only'}
VAR_GLOBAL CONSTANT
	_PER : STRING := 'per';
    _SQUARED : STRING := 'squared';
    _CUBED : STRING := 'cubed';
    _PEAK : STRING := 'peak';
    _MEGA : STRING := 'mega';
    _KILO : STRING := 'kilo';
    _CENTI : STRING := 'centi';
    _HECTO : STRING := 'hecto';
    _MICRO : STRING := 'micro';
    _MILLI : STRING := 'milli';
    _PERCENTAGE : STRING := 'percentage';
    _ACRE : STRING := 'acre';
    _HECTARE : STRING := 'hectare';
    _DECIBEL : STRING := 'decibel';
    _DECIBEL_ATTENUATED : STRING := 'decibel_attenuated';
    _KNOT : STRING := 'knot';
    _CELSIUS : STRING := 'celsius';
    _KELVIN : STRING := 'kelvin';
    _FAHRENHEIT : STRING := 'fahrenheit';
    _YEAR : STRING := 'year';
    _MONTH : STRING := 'month';
    _WEEK : STRING := 'week';
    _DAY : STRING := 'day';
    _HOUR : STRING := 'hour';
    _MINUTE : STRING := 'minute';
    _SECOND : STRING := 'second';
    _METRE : STRING := 'metre';
    _INCH : STRING := 'inch';
    _FOOT : STRING := 'foot';
    _YARD : STRING := 'yard';
    _MILE : STRING := 'mile';
    _MILE_SCANDINAVIAN : STRING := 'mile_scandinavian';
    _GRAM : STRING := 'gram';
    _OUNCE : STRING := 'ounce';
    _POUND : STRING := 'pound';
    _STONE : STRING := 'stone';
    _DEGREE : STRING := 'degree';
    _RADIAN : STRING := 'radian';
    _LITRE : STRING := 'litre';
    _GALLON : STRING := 'gallon';
    _FLUID_OUNCE : STRING := 'fluid_ounce';
    _JOULE : STRING := 'joule';
    _BTU : STRING := 'btu';
    _WATT : STRING := 'watt';
    _LUX : STRING := 'lux';
    _LUMEN : STRING := 'lumen';
    _PASCAL : STRING := 'pascal';
    _BAR : STRING := 'bar';
    _INCH_MERCURY : STRING := 'inch_mercury';
    _VOLT : STRING := 'volt';
    _OHM : STRING := 'ohm';
    _AMP : STRING := 'amp';
    _HERTZ : STRING := 'hertz';
    _RPM : STRING := 'rpm';
    _PPM : STRING := 'ppm';
    _CARBON : STRING := 'carbon';
    _VAR : STRING := 'var';
END_VAR

// ---- POUs/Objects/PowerQualityMonitor/FB_Janitza_UMG801/PowerMeterConfig.TcGVL
{attribute 'qualified_only'}
VAR_GLOBAL CONSTANT
	IP_JANITZA: STRING(16) := '192.168.1.41';
	MBPort_Janitza : UINT := 502;
END_VAR

// ---- POUs/Objects/CoolingSystem/HeatpumpSystem/IF_Heatpump.TcIO
INTERFACE IF_Heatpump

METHOD AllowMBComm : BOOL
VAR_INPUT
	b_AllowComm	:	Bool;
END_VAR
END_METHOD

METHOD EMStop : BOOL
VAR_INPUT
END_VAR
END_METHOD

METHOD getDiagnostics
VAR_IN_OUT
	AddError		: ARRAY [*] OF FB_AddErrorST;
	a_ActiveEvents	: ARRAY [*] OF ST_ErrorStruct;
	w_Index			: WORD;
END_VAR

VAR_OUTPUT
	b_errorActive	: BOOL;
	b_warningActive	: BOOL;
END_VAR
END_METHOD

METHOD MBCommBusy : BOOL
VAR_INPUT
END_VAR
END_METHOD

METHOD Reset : BOOL
VAR_INPUT
END_VAR
END_METHOD

METHOD Setpoint : BOOL
VAR_INPUT
	OperatingMode	:	eHeatpumpMode	:= 	eHeatpumpMode.Standby;
	Temperature		: 	REAL			:=	18;
END_VAR
END_METHOD

END_INTERFACE

// ---- POUs/MAIN_Fast.TcPOU
PROGRAM MAIN_Fast
VAR
	Router														: FB_Teltonika;
	SystemControl												: FB_SystemControl;
	AcDcCharger													: FB_AcDcCharger;
	ACswitchgear												: FB_ACSwitchgear;
	DCswitchgear												: FB_DCswitchgear;
	HartingIO													: FB_HartingIO;
	NeutralTransformer											: FB_NeutralTransformer;
	Coolingsystem												: FB_Coolingsystem;
	PowerStack													: FB_PowerStack;
	PowerMonitor												: FB_PowerQualityMonitoring;
	InternalPowerSupply											: FB_InternalPowerSupply;
	BMS															: FB_BMS;
	ProtectionSystems											: FB_ProtectionSystems;
	Enclosure													: FB_enclosure;
	PLCstate													: FB_PLCState;
	Peakshavebox												: FB_peakshavebox;
	GenComm														: FB_GenComm;				
END_VAR

VAR // structures containing all system control/monitoring vars and are exchanged with other task.
	{ attribute 'TcHmiSymbol.Hide' }
	monitor						: ST_System_Monitor;
	{ attribute 'TcHmiSymbol.Hide' }
	control						: REFERENCE TO ST_System_Control;

	fb_WritePersistentData		: WritePersistentData;
END_VAR

VAR
	//Reset function
	b_ResetManual			: BOOL;
	ton_EMstopTimeOut		: TON := (PT:= T#30S);
	w_MethodFbs				: WORD;
	tp_ResetDuration		: TP := (PT:= T#2S);
	ton_ForceShutdown		: ton := (PT := T#10S);
	ton_shutdownDelay		: ton := (PT := T#3S);
	b_shutdownInitiated		: BOOL;
	ton_NUCshutdownDelay	: ton := (PT := T#20S);
	
	//Method feedbacks
	EMstopFb				: BYTE;		
	b_EMstopCompleted		: BOOL;
	b_shutdownCompleted		: BOOL;
	b_MethodStartFB			: BOOL;
	r_trigInitialReset		: R_TRIG;
END_VAR

control REF= MAIN_Slow.control;

WearLogging();
SetConfig();
SetSystemMonitorControlvars();
BMS.Init();	//init method to initialize persistent variables from wearlogging

IF __ISVALIDREF(control) THEN

	PLCstate();
	
	Safety(b_extEmstopTrigger := SystemControl.toSystem.control.b_EMStop,
		b_enable := GVL.b_SystemReady
		);
		Safety.EDMSignals.b_NetcontactorEDM := Powerstack.b_NetcontEDM;
		Safety.EDMSignals.b_MccbMasterEDM:= Powerstack.b_MasterMccbEDM;
		Safety.EDMSignals.b_MccbSlaveEDM:= Powerstack.b_SlaveMccbEDM;
		
	//call FB
	
	PowerStack(
			e_ACRotationStateExt			:= powermonitor.get.OutputField.e_ACrotationStatus,
			r_PLossInternal					:= powermonitor.get.InternalSupply.ar_ActivePower[0],
			r_QLossInternal					:= powermonitor.get.InternalSupply.ar_ReactivePower[0],
			st_params						:= settings.MachineParams.Powerstack,
			st_calibration 					:= settings.Calibration.Powerstack,
			set								:= SystemControl.toSystem.Powerstack,
			b_transportMode					:= systemcontrol.toSystem.b_TransportMode,
			b_DoublePowermodule				:= settings.Configuration.b_DoublePowerModule,
			by_coolingPowerRequest			:= coolingsystem.by_PSPowerRequest,
			b_BatteryDCReady				:= BMS.PowerStatus = eHVDC_Powerstatus.ON,
			r_BatteryDCvoltage				:= BMS.get.MBMU.BatteryStatus.r_SystemVoltage,
			b_RotationswitchEnable			:= settings.Configuration.b_AutomaticACrotation,
			b_ExtgridCodeTrip				:= Powermonitor.get.OutputField.r_CurrentUnbalance > settings.GridParams.r_CurrentUnbalanceLimit AND Powermonitor.get.OutputField.ar_Current[0] > 20 AND NOT settings.Configuration.b_NeutralTransformer,
			b_EnableFan						:= coolingsystem.b_FanPowerstackEnable,
			b_OutputConnected				:= ACswitchgear.get.b_OutputMCCBfb,
			b_InputConnected				:= ACswitchgear.get.b_inputMCCBfb,// AND ACswitchgear.get.b_InputContactorfb
			b_InternalACRequired			:= InternalPowerSupply.b_PowerStackACRequired
		);

	PowerMonitor(
		b_enable:= TRUE,
		powerstackGet := powerstack.get,
		b_TNModeActive:= Monitor.protections.Insulation.e_EarthingSystemDetected <> eEarthingsystems.IT,
		b_thirdOutputfieldAvailable := settings.Configuration.b_ThirdOutputConnection,
		b_NeutralTransformerAvailable := settings.Configuration.b_NeutralTransformer,
		b_InputFieldsAvailable := settings.Configuration.b_ACInputConnection
		);
	
	InternalPowerSupply(
			st_PowerstackDemandSupply := Powerstack.st_InternalPsuSupplyRequest, 
			st_CoolingDemandSupply := Coolingsystem.IPSRequest,
			b_BusbarACAvailable := powerstack.get.b_ACdetected,
			b_PowerstackACavailable := powerstack.b_InternalPsuACOk,
			st_params:=Settings.MachineParams.Interpowersupply,
			e_BMSPowerState := BMS.PowerStatus,
			b_ConditioningOnBatteryAllowed := BMS.b_InternalHVDCAllowed
		);

	BMS(
		st_params 		:= settings.MachineParams.BMS,
		b_HVDCEnable	:= Internalpowersupply.b_HVDC_Enable,
		set 			:= Systemcontrol.toSystem.BMS,
		by_NoOfStrings	:= Settings.Configuration.by_NoBatteryStrings
	);	

	Enclosure(st_params := Settings.MachineParams.Enclosure, set := SystemControl.toSystem.Enclosure);
		Enclosure.ledstrip.SetMachineStatus(
			b_Error := GVL.b_QuickshutdownActive OR GVL.b_EmergencyShutdownActive OR GVL.b_NormalShutdownActive,
			b_warning := GVL.b_WarningActive,
			b_attention := NOT BMS.get.BatteryInfo.b_chargingAllowed OR NOT BMS.get.BatteryInfo.b_dischargingAllowed,
			b_Normal := BMS.PowerStatus = eHVDC_powerstatus.ON,
			b_off :=  Monitor.system.e_State = eSystemState.Transport,
			r_Soc := BMS.get.BatteryInfo.r_SOCScaled,
			r_DCcurrent := Powerstack.get.r_DCcurrent);

	CoolingSystem(
		st_params := settings.MachineParams.Coolingsystem,
		by_PSsetCooling:= powerstack.by_CoolingControl,
		b_InverterRunning:= powerstack.get.b_InverterRunning,
		r_InverterLoad := powerstack.get.r_LoadPercent,
		b_24v_Available := internalpowersupply.Get.b_24VdcAvailable,
		b_400v_Available := internalpowersupply.Get.b_400VACAvailable,
		e_400vSupplySource := internalpowersupply.Get.e_400VSupplySource,
		r_BMSAverageBattTemp := BMS.get.BatteryInfo.ar_CellTemperature[eSubvalues.Average],
		r_BMSMaxBattTemp := BMS.get.BatteryInfo.ar_CellTemperature[eSubvalues.Maximum],
		b_DehumStart := systemcontrol.toSystem.control.b_startDeHum,
		r_enclosureHumidity := enclosure.get.climate.r_Humidity,
		r_enclosureTemperature := enclosure.get.climate.r_Temperature,
		r_InverterTemp := Powerstack.get.PowermoduleMaster.r_TemperatureInverter,
		b_ConditioningOnBatteryAllowed := BMS.b_InternalHVDCAllowed
		);
		
	
	NeutralTransformer(
		b_enable:= settings.Configuration.b_NeutralTransformer,
		r_currentN := Powermonitor.get.BESS.ar_Current[phases.N],
		r_linevoltage := powermonitor.get.OutputField.ar_LineVoltage[Phases.AVG],
		r_voltageUnbalance := Powermonitor.get.Outputfield.r_VoltageUnbalance,
		b_NetcontactorFB := Powerstack.get.Netcontactor.b_NetConFb,
		st_params := settings.MachineParams.NeutralTransformer
		);
	
		
	ProtectionSystems(
		st_params := settings.MachineParams.Protections,
		powermonitor := Powermonitor.get,
		b_batteryAlarm := BMS.get.Events.b_OVER_TEMP_ALARM
	);
		ProtectionSystems.ToInsuMon.b_MccbfbMaster := Powerstack.get.PowermoduleMaster.b_MccbFb;
		ProtectionSystems.ToInsuMon.b_MccbfbSlave := Powerstack.get.PowermoduleSlave.b_MccbFb;
		ProtectionSystems.ToInsuMon.b_NetContFB := Powerstack.get.Netcontactor.b_NetConFb;
		ProtectionSystems.ToInsuMon.b_ACdetected := Powerstack.get.b_ACdetected;
		ProtectionSystems.ToInsuMon.b_PENlinkFB := AcSwitchgear.get.b_PENlinkfb;
		ProtectionSystems.set := systemcontrol.toSystem.Protections;
		
	ACswitchgear(
		b_inputAvailable:= settings.Configuration.b_ACInputConnection,
		b_NeutralTransformerAvailable := settings.Configuration.b_NeutralTransformer, 
		b_MCCBinputShuntTrip := protectionsystems.get.OvercurrentProtection.b_InputAlarm,
		b_MCCBOutputShuntTrip:= protectionsystems.get.overcurrentprotection.b_OutputAlarm,
		b_TransportMode := Monitor.system.e_State = eSystemState.Transport,
		set := Systemcontrol.toSystem.ACSwitchgear,
		st_params := settings.MachineParams.ACswitchgear,
		);
		
	AcDcCharger(
		st_params := settings.MachineParams.ACDCCharger,
		enable:= Settings.Configuration.b_DcCharger,
		set := systemcontrol.tosystem.AcDcCharger,(*BMS := BMS.get.BatteryInfo,*) 
		r_Soc := BMS.get.BatteryInfo.r_SOCScaled, 
		r_SystemVoltage := BMS.get.BatteryInfo.r_SystemVoltage,
		r_SystemCurrent := BMS.get.BatteryInfo.r_SystemCurrent,
		r_MaxChargeCurrent := BMS.get.BatteryInfo.r_MaxChargeCurrentAllowed,
		b_BatteryOn := (BMS.get.BatteryInfo.e_BMS_PowerOnStatus = ePowerOnSTatus.On), 
		b_BatteryFullyCharged := (BMS.get.BatteryInfo.e_BMS_Status = eBMS_status.FullCharge)
		);
		
	
	HartingIO(
		st_params := settings.MachineParams.HartingIO,
		set := systemcontrol.toSystem.HartingIO,
		SystemOperating := Powerstack.get.b_StartedState,
		SystemEmStop := Monitor.system.e_State = eSystemState.EMstop,
		);
		
	GenComm(
		st_params := settings.MachineParams.GenComm,
		set := systemcontrol.toSystem.GenComm);
	
	//external measurement box (PSB)	
	Peakshavebox(st_params := settings.MachineParams.PSB,
		b_enable:= settings.Configuration.b_PeakshaverBoxEnable AND Control.SoftSettings.setup.b_PeakshaveBoxEnable);
	PeakshaveBox.set := systemcontrol.toSystem.Peakshavebox;

	
	//Router --> GPS, 4G, SMS etc.
	Router(s_message := errorhandling.a_SMSEventBuffer, 
		st_params := Settings.MachineParams.Router,
		s_SerialNumber := settings.Properties.s_SerialNumber);
	monitor.system.b_SMSnumberConfigured := Router.SetSMSNumber(control.SoftSettings.system.s_SMSnumber);
	monitor.system.b_CustomNameConfigured:= Router.SetDevName(control.SoftSettings.system.s_SystemName);

	//FB with connection from user to system vars
	SystemControl(
		st_params := settings.MachineParams.system,
		st_calibration := settings.Calibration,
		monitor:= monitor, control:= control);
	

//CALL MAIN FUNCTIONS
	Reset(SystemControl.toSystem.control.b_Reset, NOT GVL.b_SystemReady OR settings.MachineParams.system.b_VDLReset);
	MainSFC();
	//System shutdown --> manually or by firesystem
	SystemShutdown(Systemcontrol.toSystem.control.b_SystemShutdown OR ProtectionSystems.b_SystemShutdownCMD);
END_IF

ACTION _aErrorSequence_entry:
SFCReset := TRUE;
END_ACTION

ACTION _aInit_active:
//INIT state
b_EMstopCompleted :=  FALSE;
Monitor.system.e_State:= eSystemState.Init;
END_ACTION

ACTION _aStandBy_active:
Powerstack.Standbycmd();
Internalpowersupply.HVDC_Enable();

IF systemcontrol.toSystem.b_TransportMode THEN
	IF Coolingsystem.Shutdown() THEN
		powerstack.Shutdowncmd();
	END_IF
	AcSwitchgear.set.b_inputContactorOpen := TRUE;
	Monitor.system.e_State:= eSystemState.Transport;
ELSE
	Monitor.system.e_State:= eSystemState.Init;
	Coolingsystem.Start();
	IF coolingsystem.Get.CoolingSystemMode = eCoolingSystemState.EnclosureConditioning OR 
	coolingsystem.Get.CoolingSystemMode = eCoolingSystemState.BatteryConditioning OR
	coolingsystem.Get.CoolingSystemMode = eCoolingSystemState.InverterConditioning THEN
		Monitor.system.e_State:= eSystemState.Conditioning;
	ELSIF coolingsystem.Get.CoolingSystemMode = eCoolingSystemState.DeHum OR
	coolingsystem.Get.CoolingSystemMode = eCoolingSystemState.DehumEnding THEN
		Monitor.system.e_State := eSystemState.Dehumidifying;	 
	ELSE
		Monitor.system.e_State:= eSystemState.StandBy;
	END_IF
END_IF
END_ACTION

ACTION a_ContinousActions:
ErrorSFC();
END_ACTION

ACTION a_EmergencyShutdown_active:
SFCReset := TRUE;
b_EMstopCompleted := EMStop();
Monitor.system.e_State := eSystemState.EMstop;
InternalPowersupply.HVDC_disable();
END_ACTION

ACTION a_ErrorSequence_active:
// SFC IDENTIFICATION
Powerstack.Shutdowncmd();
Reset(FALSE, systemcontrol.toSystem.control.b_Reset);

IF GVL.b_EmergencyShutdownActive THEN
	InternalPowersupply.HVDC_disable();
	Monitor.system.e_State := eSystemState.EMstop;
END_IF
END_ACTION

ACTION a_ErrorSequence_exit:
//RELEASE MAINSEQUENCE AFTER ALL ERROR ARE CLEARED
Reset(FALSE, FALSE);
SFCReset := FALSE;
END_ACTION

METHOD PUBLIC CheckDCcurrent : BOOL
VAR_INPUT
	r_in			: REAL;
END_VAR
//checkcurrent is below limit.
CheckDCcurrent := (BMS.get.BatteryInfo.r_SystemCurrent < r_in AND powerstack.get.r_DCcurrent < r_in);
END_METHOD

METHOD EMstop : BOOL

VAR
	EMstopDone	: BOOL;
END_VAR
//EMstopDone := Powerstack.EMstop() AND 
//	Coolingsystem.EMSTOP() AND 
//	Internalpowersupply.EMstop() AND 
//	BMS.EMSTOP() AND 
//	systemcontrol.EMstop();
	
EMstopFb.0 := Powerstack.EMstop();
EMstopFb.1 := Coolingsystem.EMSTOP();
EMstopFb.2 := Internalpowersupply.EMstop();
EMstopFb.3 := BMS.EMSTOP();
EMstopFb.4 := systemcontrol.EMstop();
EMstopFb.5 := ACDCCharger.EMSTOP();;
EMstopFb.6 := TRUE;
EMstopFb.7 := TRUE;

EMstopDone:= EMstopFb = 255;

ton_EMstopTimeOut(IN:= NOT EMstopDone);
EMstop := EMstopDone; //OR ton_EMstopTimeOut.Q;

IF EMstopDone THEN
	EMstopFb := 0;
END_IF

//IF ton_EMstopTimeOut.Q THEN
//	InternalPowersupply.SystemShutdown(FALSE);
//END_IF
END_METHOD

ACTION ErrorSFC:
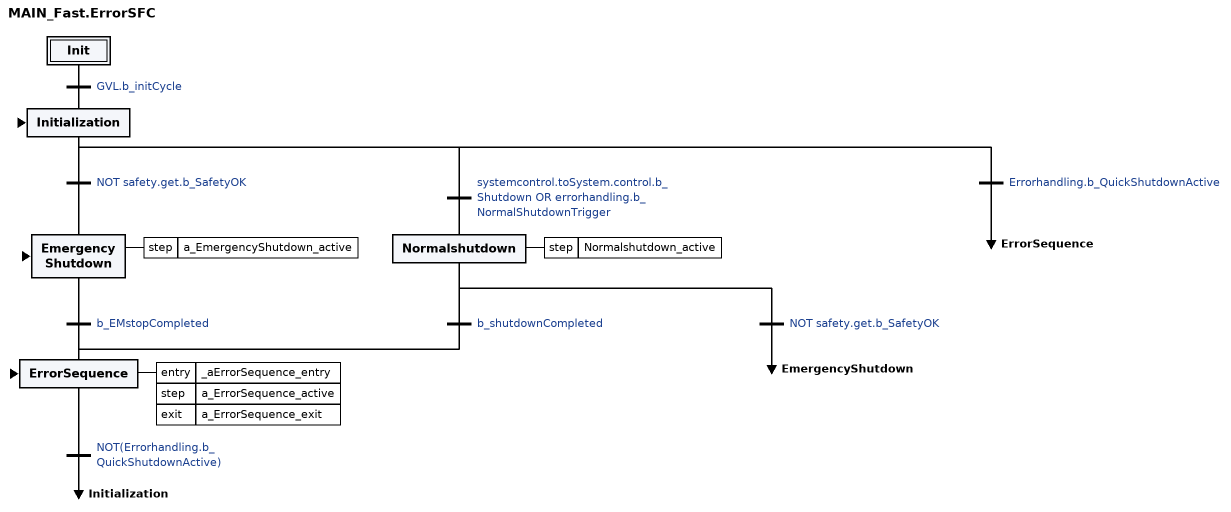
INITIAL_STEP Init:
END_STEP
TRANSITION FROM Init TO Initialization
    := GVL.b_initCycle;
END_TRANSITION
STEP Initialization:
END_STEP
TRANSITION FROM Initialization TO EmergencyShutdown
    := NOT safety.get.b_SafetyOK;
END_TRANSITION
STEP EmergencyShutdown:
    a_EmergencyShutdown_active(N);  // step action
END_STEP
TRANSITION FROM EmergencyShutdown TO ErrorSequence
    := b_EMstopCompleted;
END_TRANSITION
TRANSITION FROM Initialization TO Normalshutdown
    := systemcontrol.toSystem.control.b_Shutdown OR errorhandling.b_NormalShutdownTrigger;
END_TRANSITION
STEP Normalshutdown:
    Normalshutdown_active(N);  // step action
END_STEP
TRANSITION FROM Normalshutdown TO ErrorSequence
    := b_shutdownCompleted;
END_TRANSITION
TRANSITION FROM Normalshutdown TO EmergencyShutdown
    := NOT safety.get.b_SafetyOK;
END_TRANSITION
TRANSITION FROM Initialization TO ErrorSequence
    := Errorhandling.b_QuickShutdownActive;
END_TRANSITION
STEP ErrorSequence:  // min time T#5s
    _aErrorSequence_entry(P1);  // entry action
    a_ErrorSequence_active(N);  // step action
    a_ErrorSequence_exit(P0);  // exit action
END_STEP
TRANSITION FROM ErrorSequence TO Initialization
    := NOT(Errorhandling.b_QuickShutdownActive);
END_TRANSITION
// branch label Branch1_ErrorSFC
// branch label Branch0_ErrorSFC
END_ACTION

ACTION IdleOperation_active:
IF powerstack.stopcmd() THEN
	Monitor.system.e_State := eSystemState.Stopped;
END_IF
END_ACTION

ACTION InitializeMachine_active:

END_ACTION

ACTION MainSFC:
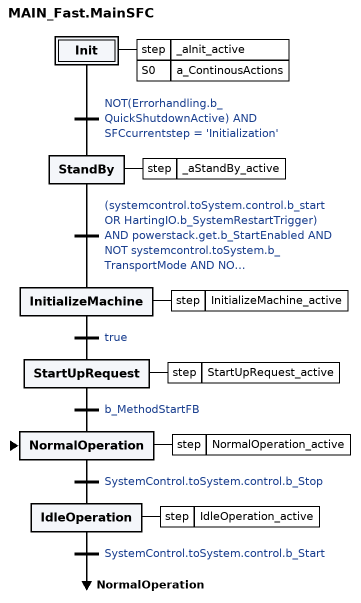
INITIAL_STEP Init:
    _aInit_active(N);  // step action
    a_ContinousActions(S0);
END_STEP
TRANSITION FROM Init TO StandBy
    := NOT(Errorhandling.b_QuickShutdownActive) AND SFCcurrentstep = 'Initialization';
END_TRANSITION
STEP StandBy:
    _aStandBy_active(N);  // step action
END_STEP
TRANSITION FROM StandBy TO InitializeMachine
    := (systemcontrol.toSystem.control.b_start OR HartingIO.b_SystemRestartTrigger) AND powerstack.get.b_StartEnabled AND NOT systemcontrol.toSystem.b_TransportMode AND NOT GVL.b_NormalShutdownActive;
END_TRANSITION
STEP InitializeMachine:
    InitializeMachine_active(N);  // step action
END_STEP
TRANSITION FROM InitializeMachine TO StartUpRequest
    := true;
END_TRANSITION
STEP StartUpRequest:
    StartUpRequest_active(N);  // step action
END_STEP
TRANSITION FROM StartUpRequest TO NormalOperation
    := b_MethodStartFB;
END_TRANSITION
STEP NormalOperation:
    NormalOperation_active(N);  // step action
END_STEP
TRANSITION FROM NormalOperation TO IdleOperation
    := SystemControl.toSystem.control.b_Stop;
END_TRANSITION
STEP IdleOperation:
    IdleOperation_active(N);  // step action
END_STEP
TRANSITION FROM IdleOperation TO NormalOperation
    := SystemControl.toSystem.control.b_Start;
END_TRANSITION
END_ACTION

ACTION NormalOperation_active:
powerstack.startcmd();

IF powerstack.get.e_State = eStatusPowerstack.running THEN
	IF NOT bms.get.BatteryInfo.b_chargingAllowed THEN
		Monitor.system.e_State := eSystemState.Discharging_Only;
	ELSIF NOT bms.get.BatteryInfo.b_DischargingAllowed THEN
		Monitor.system.e_State := eSystemState.Charging_Only;
	ELSE
		Monitor.system.e_State := eSystemState.Running;
	END_IF
ELSE
	IF powerstack.get.e_State = eStatusPowerstack.idle OR powerstack.get.e_State = eStatusPowerstack.GridCodeStop THEN
		Monitor.system.e_State := eSystemState.Stopped;	
	ELSE
		Monitor.system.e_State := eSystemState.Starting;	
	END_IF	
END_IF
END_ACTION

ACTION Normalshutdown_active:
SFCReset := TRUE;
b_shutdownCompleted := Powerstack.Shutdowncmd();
Monitor.system.e_State := eSystemState.shutdown;
END_ACTION

METHOD PUBLIC Reset : BOOL
VAR_INPUT
	b_reset	: BOOL;
	b_force : BOOL;
END_VAR
tp_ResetDuration(IN := b_reset OR b_Force);

//reinitiliaze reset statuss if reset is retriggered
IF tp_resetDuration.Q = FALSE THEN
	w_MethodFbs := 0;
END_IF


//Everything that is not automatically reset
IF tp_ResetDuration.Q AND w_MethodFbs <> 16#FF THEN
	monitor.system.e_State := eSystemState.Reset;
	
	IF NOT w_MethodFbs.0 AND b_force THEN w_MethodFbs.0 := Safety.Reset(TRUE); END_IF
	IF NOT w_MethodFbs.1 THEN w_MethodFbs.1 := InternalPowerSupply.Reset(); END_IF
	IF NOT w_MethodFbs.2 THEN w_MethodFbs.2 := Powerstack.Reset(); END_IF
	IF NOT w_MethodFbs.3 THEN w_MethodFbs.3 := protectionSystems.Reset(); END_IF
	IF NOT w_MethodFbs.4 THEN w_MethodFbs.4 := Powermonitor.Reset(); END_IF 
	IF NOT w_MethodFbs.5 THEN w_MethodFbs.5 := BMS.Reset(); END_IF 
	IF NOT w_MethodFbs.6 THEN w_MethodFbs.6 := Neutraltransformer.Reset(); END_IF
	IF NOT w_MethodFbs.7 THEN w_MethodFbs.7 := Coolingsystem.Reset(); END_IF
	IF NOT w_MethodFbs.8 THEN w_MethodFbs.8 := Router.Reset(); END_IF
	IF NOT w_MethodFbs.9 THEN w_MethodFbs.9	:= systemcontrol.Reset(); END_IF
	IF NOT w_MethodFbs.10 THEN w_MethodFbs.10:= ACDCCharger.Reset(); END_IF
	IF NOT w_MethodFbs.11 THEN w_MethodFbs.11:= TRUE; END_IF
	IF NOT w_MethodFbs.12 THEN w_MethodFbs.12:= TRUE; END_IF
	IF NOT w_MethodFbs.13 THEN w_MethodFbs.13:= TRUE; END_IF
	IF NOT w_MethodFbs.14 THEN w_MethodFbs.14:= TRUE; END_IF
	IF NOT w_MethodFbs.15 THEN w_MethodFbs.15:= TRUE; END_IF
END_IF

//Everything that is automatically reset one in error state
Reset := w_MethodFbs = 255;
END_METHOD

ACTION SetConfig:
{IF defined (ePU10_360_N_DC_IO_PSB)}
	settings.Configuration.b_PeakshaverBoxEnable 	:= TRUE;
	settings.Configuration.b_DCbuscoupling 			:= FALSE; //TRUE;
	settings.Configuration.b_NeutralTransformer		:= TRUE;
	settings.Configuration.b_ACInputConnection		:= TRUE;
	settings.Properties.s_ConfigurationCode 		:= 'ePU10_360_N_DC_IO_PSB';
{END_IF}

{IF defined (ePU10_360_N_IO_PSB)}
	settings.Properties.s_ConfigurationCode 		:= 'ePU10_360_N_IO_PSB';
	settings.Configuration.b_ACInputConnection		:= TRUE;
	settings.Configuration.b_NeutralTransformer		:= TRUE;
	settings.Configuration.b_PeakshaverBoxEnable 	:= TRUE;
{END_IF}

{IF defined (ePU10_360_N_IO)}
	settings.Properties.s_ConfigurationCode 		:= 'ePU10_360_N_IO';
	settings.Configuration.b_ACInputConnection		:= TRUE;
	settings.Configuration.b_NeutralTransformer		:= TRUE;
{END_IF}

{IF defined (ePU10_368_3P_O_PSB)}
	settings.Properties.s_ConfigurationCode 		:= 'ePU10_368_3P_O_PSB';
	settings.Configuration.b_PeakshaverBoxEnable 	:= TRUE;
{END_IF}

{IF defined (ePU10_360_3P_O)}
	settings.Properties.s_ConfigurationCode 		:= 'ePU10_360_3P_O';
{END_IF}

IF enclosure.get.ledstrip.BeckhoffLed AND FIND(settings.Properties.s_ConfigurationCode,'_BL') = 0 THEN
	settings.Properties.s_ConfigurationCode := CONCAT(settings.Properties.s_ConfigurationCode, '_BL');
END_IF

settings.Properties.by_SWverMajor	:=	1;	
settings.Properties.by_SWverMinor	:=	6;	
settings.Properties.by_SWverPatch	:=	1;	
settings.Properties.by_SWverBuild	:=	1;	

//Set properties
settings.Properties.s_SWversionNumber				:= 	concat('V', TO_STRING(settings.Properties.by_SWverMajor));
settings.Properties.s_SWversionNumber				:=	concat(settings.Properties.s_SWversionNumber, '.');
settings.Properties.s_SWversionNumber				:= 	concat(settings.Properties.s_SWversionNumber, TO_STRING(settings.Properties.by_SWverMinor));
settings.Properties.s_SWversionNumber				:=	concat(settings.Properties.s_SWversionNumber, '.');
settings.Properties.s_SWversionNumber				:= 	concat(settings.Properties.s_SWversionNumber, TO_STRING(settings.Properties.by_SWverPatch));
IF settings.Properties.by_SWverBuild > 0 THEN
	settings.Properties.s_SWversionNumber				:=	concat(settings.Properties.s_SWversionNumber, '_');
	settings.Properties.s_SWversionNumber				:= 	concat(settings.Properties.s_SWversionNumber, TO_STRING(settings.Properties.by_SWverBuild));
END_IF
	
settings.Properties.r_RatedEnergyCapacity 			:= BMS.get.BatteryInfo.r_ratedEnergyCapacity;
settings.Properties.r_RatedActivePower 				:= MIN(BMS.get.BatteryInfo.r_ratedPower, powerstack.get.r_ratedPower);
settings.Properties.r_RatedApparentPower			:= TO_INT(powerstack.get.r_RatedCurrent * 400 * 1.73 / 1000);
settings.Properties.r_Ratedcurrent 					:= powerstack.get.r_RatedCurrent;
settings.Properties.r_ratedCurrentInput				:= SEL(settings.Configuration.b_ACInputConnection, 0, 700);
settings.Properties.r_ratedCurrentOutput			:= SEL(settings.Configuration.b_ThirdOutputConnection, 800, 1200);


CASE settings.Configuration.by_NoBatteryStrings OF
	2: settings.Properties.s_Weight					:= '7000 kg';
	3: settings.Properties.s_Weight					:= '8500 kg';
	4: settings.Properties.s_Weight					:= '9500 kg';
END_CASE
END_ACTION

ACTION SetSystemMonitorControlvars:
//First bind references
Monitor.safety := Safety.get;
Monitor.powerstack REF= Powerstack.get;
Monitor.AcDcCharger REF= AcDcCharger.get;
Monitor.powermonitor REF= Powermonitor.get;
Monitor.neutraltransformer REF= neutraltransformer.get;
Monitor.protections REF= ProtectionSystems.get;
Monitor.battery REF= BMS.get;
Monitor.ACswitchgear REF= ACswitchgear.get;
Monitor.DCswitchgear REF= DCswitchgear.get;
Monitor.peakshavebox REF= Peakshavebox.get;
Monitor.enclosure REF= Enclosure.get;
Monitor.internalpsu REF= Internalpowersupply.Get;
Monitor.PLC REF= PLCstate.get;
Monitor.Cooling REF= coolingsystem.Get;
Monitor.Router REF= Router.Get;
Monitor.Generator REF= Gencomm.Get;
Monitor.HartingIO REF= HartingIO.Get;
END_ACTION

ACTION StartUpRequest_active:
b_MethodStartFB	:= Powerstack.Startcmd();
Monitor.system.e_State:= eSystemState.Starting;
END_ACTION

METHOD SystemShutdown : BOOL
VAR_INPUT
	b_execute			: BOOL;
END_VAR
//write persisten data
fb_WritePersistentData(NETID := '', PORT:= 851, START:=b_execute,  TMOUT := T#5S);

//set force shutdown timer
ton_ForceShutdown(IN:= b_execute);
ton_shutdownDelay(IN:= b_execute);

IF ton_shutdownDelay.Q THEN
	b_shutdownInitiated := TRUE;
END_IF

//Everything that is not automatically reset
IF b_shutdownInitiated THEN
	settings.Save := TRUE;
	Monitor.system.e_State := eSystemState.shutdown;
	IF NOT w_MethodFbs.0 THEN w_MethodFbs.0 := Powerstack.Shutdowncmd(); END_IF	
	IF NOT w_MethodFbs.1 THEN w_MethodFbs.1 := SystemControl.shutdown(); END_IF
	IF NOT w_MethodFbs.2 THEN w_MethodFbs.2 := CoolingSystem.shutdown(); END_IF;
	w_MethodFbs.3 := TRUE;	
	w_MethodFbs.4 := TRUE; 
	w_MethodFbs.5 := TRUE; 
	w_MethodFbs.6 := TRUE; 
	w_MethodFbs.7 := TRUE;
ELSE
	w_MethodFbs := 0;
END_IF

IF w_MethodFbs = 255 OR ton_ForceShutdown.Q THEN
	settings.Save := FALSE;
	MqttComOpenRemote.shutdown();
	ton_NUCshutdownDelay(IN:=TRUE);
	IF ton_NUCshutdownDelay.Q THEN
		Monitor.system.e_State := eSystemState.off;
		InternalPowerSupply.SystemShutdown(timedshutdown := FALSE);
		b_shutdownInitiated := FALSE;
	END_IF
END_IF
END_METHOD

END_PROGRAM

// ---- POUs/Objects/4Grouter/FB_Teltonika.TcPOU
FUNCTION_BLOCK FB_Teltonika

VAR_IN_OUT CONSTANT
	st_params	: st_Router_Params;
END_VAR

VAR
	realconverter : dwtoreal;
	w_SendSMS: WORD;
	set : st_router_set;
	ui_counter	:	uint;
END_VAR
VAR_OUTPUT
	Get	:	st_router_get;
END_VAR
VAR
	MBRead			: 	FB_MBReadRegs;
	MBWrite			:	FB_MBWriteRegs;
	MBSingleWrite	:	FB_MBWriteSingleReg;
	
	arw_DataBuffer		: 	ARRAY[0..62] OF word;
	st_WriteSMSData		:	STRING(20);

	ar_SMSData			:	ARRAY[0..89] OF WORD;
	ar_ReadSMSData		:	ARRAY[0..89] OF WORD;
	
	tempbuffer			:	ARRAY[0..10] OF WORD;

	
	ton_GetDataTimer				:	TON := (PT := TIME#1000MS);
	ton_StartSMSServiceDelay		:	TON := (PT := T#60S);

	
	ftrig_TransmissionDone	:	F_trig;
	
	ui_MBRetryCount			:	UINT;
	ui_SMSRetryCounter	:	UINT;
		
	ui_ForCounter	:	UINT;
	ui_MessageCounter	:	UINT;
	b_busy: BOOL;
	b_CommError: BOOL;
	udi_errid: UDINT;
	udi_cbread: UDINT;
	
	
	TempDTString	:	String;
END_VAR


VAR_IN_OUT
	s_Message	:	ARRAY[*] OF STRING;
END_VAR

VAR_INPUT
	s_SerialNumber		: STRING;
END_VAR

VAR CONSTANT
	e_ID 				: eObject_ID := eObject_ID.Router;
END_VAR

ton_GetDataTimer(IN:=NOT ton_GetDataTimer.Q);
ton_StartSMSServiceDelay();

ReadDataSFC();

get.Events.b_MBCommWarning := ui_MBRetryCount > 20;


//temporary setup via stparams until hmi setup is implemented.
set := st_params.ManualSettings;

ACTION aCheckAlarmMessages:
IF ton_StartSMSServiceDelay.Q THEN
	IF get.e_SMSStatus = eSMSStatus.Idle OR get.e_SMSStatus = eSMSStatus.error THEN
		//skip through message array until non_empty value or the end of the list is found 
		WHILE (s_Message[ui_MessageCounter] = '') AND (ui_MessageCounter < UPPER_BOUND(s_message, 1)) DO
			ui_MessageCounter := ui_MessageCounter + 1;
		END_WHILE
		
		IF (s_Message[ui_MessageCounter] <> '') THEN
			CreateMessage(s_Message[ui_MessageCounter]);	//check for valid message
			get.e_SMSStatus := eSMSStatus.NewMessage;
			s_Message[ui_MessageCounter] := '';
		END_IF
		
		IF ui_MessageCounter >= UPPER_BOUND(s_message, 1) THEN
			ui_MessageCounter := DINT_TO_UINT(LOWER_BOUND(s_message, 1)); 
		END_IF
	END_IF
END_IF
END_ACTION

ACTION aNetworkinfo:
MBRead(
	sIPAddr := st_params.IP_TELTONIKA,
	nTCPPort := st_params.MBPort_TELTONIKA,
	nUnitID := 1,
	nMBAddr := 103,
	nQuantity := 32,//*2,
	cbLength := SIZEOF(arw_DataBuffer),
	pDestAddr := ADR(arw_DataBuffer),
	bExecute := ton_GetDataTimer.Q,
	bBusy => b_busy,
	bError => b_CommError,
	nErrId => udi_errid,
	cbRead => udi_cbread,
	tTimeout := st_params.T_MBTimeout
);

ftrig_TransmissionDone(clk := b_busy);

IF ftrig_TransmissionDone.q THEN
	IF NOT b_CommError THEN
		FOR ui_ForCounter := 0 TO 31 DO
			arw_DataBuffer[ui_ForCounter] := be16_TO_HOST(arw_DataBuffer[ui_ForCounter]);
		END_FOR
		
		MEMCPY(ADR(Get.Mobile.NetworkInfo),  ADR(arw_DataBuffer[0]), 32);
		MEMCPY(ADR(Get.Mobile.NetworkType),  ADR(arw_DataBuffer[16]), 32);
		ui_MBRetryCount := 0;
		sfctip := TRUE;
	ELSE
		ui_MBRetryCount := ui_MBRetryCount + 1;
		sfctip := TRUE;
	END_IF
END_IF
END_ACTION

ACTION aReadActiveSim:

MBRead(
	sIPAddr := st_params.IP_TELTONIKA,
	nTCPPort := st_params.MBPort_TELTONIKA,
	nUnitID := 1,
	nMBAddr := 205,
	nQuantity := 1,//*2,
	cbLength := SIZEOF(arw_DataBuffer),
	pDestAddr := ADR(arw_DataBuffer),
	bExecute := ton_GetDataTimer.Q,
	bBusy => b_busy,
	bError => b_CommError,
	nErrId => udi_errid,
	cbRead => udi_cbread,
	tTimeout := st_params.T_MBTimeout
);

ftrig_TransmissionDone(clk := b_busy);

IF ftrig_TransmissionDone.q THEN
	IF NOT b_CommError THEN
	
		//Get.Mobile.ui_ActiveSim := arw_DataBuffer[0];
	
		ui_MBRetryCount := 0;
		sfctip := TRUE;
	ELSE
		ui_MBRetryCount := ui_MBRetryCount + 1;
		sfctip := TRUE;
	END_IF
END_IF
END_ACTION

ACTION aReadDataUsageSim1:

MBRead(
	sIPAddr := st_params.IP_TELTONIKA,
	nTCPPort := st_params.MBPort_TELTONIKA,
	nUnitID := 1,
	nMBAddr := 193,
	nQuantity := 4,//*2,
	cbLength := SIZEOF(arw_DataBuffer),
	pDestAddr := ADR(arw_DataBuffer),
	bExecute := ton_GetDataTimer.Q,
	bBusy => b_busy,
	bError => b_CommError,
	nErrId => udi_errid,
	cbRead => udi_cbread,
	tTimeout := st_params.T_MBTimeout
);

ftrig_TransmissionDone(clk := b_busy);

IF ftrig_TransmissionDone.q THEN
	IF NOT b_CommError THEN
	
		MEMCPY(ADR(Get.Mobile.ui_Sim1DataReceivedMonth)+2, ADR(arw_DataBuffer[0]), 2);
		MEMCPY(ADR(Get.Mobile.ui_Sim1DataReceivedMonth), ADR(arw_DataBuffer[1]), 2);
		
		MEMCPY(ADR(Get.Mobile.ui_Sim1DataSendMonth)+2, ADR(arw_DataBuffer[2]), 2);
		MEMCPY(ADR(Get.Mobile.ui_Sim1DataSendMonth), ADR(arw_DataBuffer[3]), 2);	
	
		ui_MBRetryCount := 0;
		sfctip := TRUE;
	ELSE
		ui_MBRetryCount := ui_MBRetryCount + 1;
		sfctip := TRUE;
	END_IF
END_IF
END_ACTION

ACTION aReadDataUsageSim2:

MBRead(
	sIPAddr := st_params.IP_TELTONIKA,
	nTCPPort := st_params.MBPort_TELTONIKA,
	nUnitID := 1,
	nMBAddr := 308,
	nQuantity := 4,//*2,
	cbLength := SIZEOF(arw_DataBuffer),
	pDestAddr := ADR(arw_DataBuffer),
	bExecute := ton_GetDataTimer.Q,
	bBusy => b_busy,
	bError => b_CommError,
	nErrId => udi_errid,
	cbRead => udi_cbread,
	tTimeout := st_params.T_MBTimeout
);

ftrig_TransmissionDone(clk := b_busy);

IF ftrig_TransmissionDone.q THEN
	IF NOT b_CommError THEN
	
		MEMCPY(ADR(Get.Mobile.ui_Sim2DataReceivedMonth)+2, ADR(arw_DataBuffer[0]), 2);
		MEMCPY(ADR(Get.Mobile.ui_Sim2DataReceivedMonth), ADR(arw_DataBuffer[1]), 2);
		
		MEMCPY(ADR(Get.Mobile.ui_Sim2DataSendMonth)+2, ADR(arw_DataBuffer[2]), 2);
		MEMCPY(ADR(Get.Mobile.ui_Sim2DataSendMonth), ADR(arw_DataBuffer[3]), 2);	
	
		ui_MBRetryCount := 0;
		sfctip := TRUE;
	ELSE
		ui_MBRetryCount := ui_MBRetryCount + 1;
		sfctip := TRUE;
	END_IF
END_IF
END_ACTION

ACTION AReadGeneral:

MBRead(
	sIPAddr := st_params.IP_TELTONIKA,
	nTCPPort := st_params.MBPort_TELTONIKA,
	nUnitID := 1,
	nMBAddr := 1,
	nQuantity := 6,//*2,
	cbLength := SIZEOF(arw_DataBuffer),
	pDestAddr := ADR(arw_DataBuffer),
	bExecute := ton_GetDataTimer.Q,
	bBusy => b_busy,
	bError => b_CommError,
	nErrId => udi_errid,
	cbRead => udi_cbread,
	tTimeout := st_params.T_MBTimeout
);

ftrig_TransmissionDone(clk := b_busy);

IF ftrig_TransmissionDone.q THEN
	IF NOT b_CommError THEN
		
		get.Device.SystemUptime :=	SHL(	WORD_TO_UDINT(	arw_DataBuffer[0]),16)	+	arw_DataBuffer[1];
		MEMCPY(ADR(Get.Mobile.RSSI)+2,  ADR(arw_DataBuffer[2]), 2);
		MEMCPY(ADR(Get.Mobile.RSSI),  ADR(arw_DataBuffer[3]), 2);

		//MEMCPY(ADR(Get.Mobile.NetworkOperator),  ADR(arw_DataBuffer[22]), 32);
		
		get.Device.Temperature	:= 	UDINT_TO_REAL ( SHL(	WORD_TO_UDINT(	arw_DataBuffer[4]),16)	+	arw_DataBuffer[5] )/10;

		ui_MBRetryCount := 0;
		sfctip := TRUE;
	ELSE
		ui_MBRetryCount := ui_MBRetryCount + 1;
		sfctip := TRUE;
	END_IF
END_IF
END_ACTION

ACTION aReadGPSData:


MBRead(
	sIPAddr := st_params.IP_TELTONIKA,
	nTCPPort := st_params.MBPort_TELTONIKA,
	nUnitID := 1,
	nMBAddr := 143,
	nQuantity := 42,//*2,
	cbLength := SIZEOF(arw_DataBuffer),
	pDestAddr := ADR(arw_DataBuffer),
	bExecute := ton_GetDataTimer.Q,
	bBusy => b_busy,
	bError => b_CommError,
	nErrId => udi_errid,
	cbRead => udi_cbread,
	tTimeout := st_params.T_MBTimeout
);

ftrig_TransmissionDone(clk := b_busy);

IF ftrig_TransmissionDone.q THEN
	IF NOT b_CommError THEN
		
		realconverter.Registers[2] := arw_DataBuffer[0];
		realconverter.Registers[1] := arw_DataBuffer[1];
		Get.GPS.Latitude  := realconverter.realvalue;
 
		realconverter.Registers[2] := arw_DataBuffer[2];
		realconverter.Registers[1] := arw_DataBuffer[3];
		Get.GPS.Longitude  := realconverter.realvalue;
		
		FOR ui_ForCounter := 4 TO 35 DO
			arw_DataBuffer[ui_ForCounter] := be16_TO_HOST(arw_DataBuffer[ui_ForCounter]);
		END_FOR
				
		MEMCPY(ADR(Get.GPS.FixTime),  ADR(arw_DataBuffer[4]), 32);			//GPS fixtime (text, unix timetamp * 1000)
						
		MEMCPY(ADR(TempDTString), ADR(arw_DataBuffer[20]), 32);			//GPS DateTime (text, YYYY-MM-DD HH:MM:SS)
		FindAndReplaceChar(ADR(TempDTString), ' ', '-', ADR(TempDTString), SIZEOF(TempDTString));	//replace space between date and time with dash
		TempDTString := concat(TempDTString, '.000');	//add milliseconds to string
		get.GPS.DateTime := SystemTime_TO_DT(String_TO_Systemtime(TempDTString));
		
		realconverter.Registers[2] := arw_DataBuffer[36];					//GPS speed
		realconverter.Registers[1] := arw_DataBuffer[37];
		Get.GPS.Speed  := realconverter.realvalue;
		
	
		MEMCPY(ADR(Get.GPS.SatCount)+2, ADR(arw_DataBuffer[38]), 2);			//GPS sattelite count
		MEMCPY(ADR(Get.GPS.SatCount), ADR(arw_DataBuffer[39]), 2);			//GPS sattelite count
		
		realconverter.Registers[2] := arw_DataBuffer[40];
		realconverter.Registers[1] := arw_DataBuffer[41];
		Get.GPS.Accuracy  := realconverter.realvalue;						//GPS accuracy
		
			
		ui_MBRetryCount := 0;
		sfctip := TRUE;
	ELSE
		ui_MBRetryCount := ui_MBRetryCount + 1;
		sfctip := TRUE;
	END_IF
END_IF
END_ACTION

ACTION aReadSerial:
MBRead(
	sIPAddr := st_params.IP_TELTONIKA,
	nTCPPort := st_params.MBPort_TELTONIKA,
	nUnitID := 1,
	nMBAddr := 39,
	nQuantity := 16,//*2,
	cbLength := SIZEOF(arw_DataBuffer),
	pDestAddr := ADR(arw_DataBuffer),
	bExecute := ton_GetDataTimer.Q,
	bBusy => b_busy,
	bError => b_CommError,
	nErrId => udi_errid,
	cbRead => udi_cbread,
	tTimeout := st_params.T_MBTimeout
);

ftrig_TransmissionDone(clk := b_busy);

IF ftrig_TransmissionDone.q THEN
	IF NOT b_CommError THEN
		FOR ui_ForCounter := 0 TO 16 DO
			arw_DataBuffer[ui_ForCounter] := be16_TO_HOST(arw_DataBuffer[ui_ForCounter]);
		END_FOR
		
		//MEMCPY(ADR(Get.Mobile.NetworkOperator),  ADR(arw_DataBuffer[0]), 32);
		MEMCPY(ADR(Get.Device.RouterSerial),  ADR(arw_DataBuffer[0]), 32);
		
		ui_MBRetryCount := 0;
		sfctip := TRUE;
	ELSE
		ui_MBRetryCount := ui_MBRetryCount + 1;
		sfctip := TRUE;
	END_IF
END_IF
END_ACTION

ACTION aSendSMS:

IF get.e_SMSStatus = eSMSStatus.SendingMessage THEN
	MBSingleWrite(
		sIPAddr := st_params.IP_TELTONIKA,
		nTCPPort := st_params.MBPort_TELTONIKA,
		nUnitID := 1,
		nMBAddr := 396,
		nValue	:=	1,
		bExecute := ton_GetDataTimer.Q,
		bBusy => b_busy,
		bError => b_CommError,
		nErrId => udi_errid,
		tTimeout := st_params.T_MBTimeout
	);
	
	ftrig_TransmissionDone(clk := b_busy);
	
	IF ftrig_TransmissionDone.q THEN
		IF NOT b_CommError THEN
			get.e_SMSStatus := eSMSSTatus.idle;		
			ui_SMSRetryCounter := 0;
			ui_MBRetryCount := 0;
			sfctip := TRUE;
		ELSE
			ui_MBRetryCount := ui_MBRetryCount + 1;
			ui_SMSRetryCounter := ui_SMSRetryCounter + 1;
			IF ui_SMSRetryCounter > 0 THEN
				get.Events.b_SMSNotSendError := TRUE;
				get.e_SMSStatus := eSMSStatus.error;
				sfctip := TRUE;
			END_IF
		END_IF
	END_IF
ELSE
	SFCtip := NOT SFCTip;
END_IF
END_ACTION

ACTION aWriteSimSettings:

arw_DataBuffer[0] := TO_UINT(set.SimSelectionMode);
arw_DataBuffer[1] := TO_UINT(set.Sim1Pin);
arw_DataBuffer[2] := TO_UINT(set.Sim2Pin);

//FOR ui_counter := 1 TO 3 DO
//	arw_DataBuffer[ui_counter] := host_to_be16(arw_DataBuffer[ui_counter]);
//END_FOR

MBWrite(
	sIPAddr := st_params.IP_TELTONIKA,
	nTCPPort := st_params.MBPort_TELTONIKA,
	nUnitID := 1,
	nMBAddr := 1049,
	nQuantity := 3,
	cbLength := SIZEOF(arw_DataBuffer),
	pSrcAddr	:=	ADR(arw_DataBuffer),
	bExecute := ton_GetDataTimer.Q,
	bBusy => b_busy,
	bError => b_CommError,
	nErrId => udi_errid,
	tTimeout := st_params.T_MBTimeout
);

ftrig_TransmissionDone(clk := b_busy);

IF ftrig_TransmissionDone.q THEN
		sfctip := TRUE;
END_IF
END_ACTION

ACTION aWriteSMSData:

MBWrite(
	sIPAddr := st_params.IP_TELTONIKA,
	nTCPPort := st_params.MBPort_TELTONIKA,
	nUnitID := 1,
	nMBAddr := 397,
	nQuantity := 90,
	cbLength := SIZEOF(ar_SMSData),
	pSrcAddr	:=	ADR(ar_SMSData),
	bExecute := ton_GetDataTimer.Q,
	bBusy => b_busy,
	bError => b_CommError,
	nErrId => udi_errid,
	tTimeout := st_params.T_MBTimeout
);

ftrig_TransmissionDone(clk := b_busy);

IF ftrig_TransmissionDone.q THEN
	IF NOT b_CommError THEN
		get.e_SMSStatus := eSMSStatus.SendingMessage;
		ui_SMSRetryCounter := 0;
		ui_MBRetryCount := 0;
		sfctip := TRUE;
	ELSE
		ui_SMSRetryCounter := ui_SMSRetryCounter +1;
		ui_MBRetryCount := ui_MBRetryCount + 1;
		IF ui_SMSRetryCounter > 3 THEN
			get.Events.b_SMSNotSendError := TRUE;
			get.e_SMSStatus := eSMSStatus.error;
			sfctip := TRUE;
		END_IF
	END_IF
END_IF
END_ACTION

ACTION Bypass_active:
get.e_SMSStatus := eSMSStatus.Idle;
get.Events.b_SMSNotSendError := FALSE;
END_ACTION

METHOD CreateMessage : BOOL
VAR_INPUT
//	TelNumber	:	ULINT;
	s_Message		:	STRING(80);
END_VAR

VAR
	s_InternalMessage 	: 	STRING(160);
	s_LAT				:	STRING(8);
	s_LONG				:	STRING(9);
	ui_counter			:	UINT;
END_VAR
IF NOT get.Events.b_NoSMSNumberAvailable THEN
	memcpy(ADR(ar_SMSData[0]), ADR(get.Mobile.s_EmergencySMSNumber), 20);
	
	s_LAT := REAL_TO_STRING(get.GPS.Latitude);
	s_LONG := REAL_TO_STRING(get.GPS.Longitude);
	
	s_InternalMessage := 'ePU10 LFP Battery System';
	s_InternalMessage := concat(s_InternalMessage, '$n');
	s_InternalMessage := concat(s_InternalMessage, 'ID: ');
	s_InternalMessage := concat(s_InternalMessage, get.mobile.s_EmergencySMSDevName);
	s_InternalMessage := concat(s_InternalMessage, '$n');
	s_InternalMessage := concat(s_InternalMessage, 'LAT: ');
	s_InternalMessage := concat(s_InternalMessage, s_LAT);
	s_InternalMessage := concat(s_InternalMessage, '$n');
	s_InternalMessage := concat(s_InternalMessage, 'LON: ');
	s_InternalMessage := concat(s_InternalMessage, s_LONG);
	s_InternalMessage := concat(s_InternalMessage, '$n');
	s_InternalMessage := concat(s_InternalMessage,s_Message);
	
	memcpy(ADR(ar_SMSData[10]), ADR(s_InternalMessage[0]), 160);
	
	FOR ui_counter := 0 TO 89 DO
		ar_SMSData[ui_counter] := host_to_be16(ar_SMSData[ui_counter]);
	END_FOR

	CreateMessage := TRUE;
ELSE
	get.Events.b_SMSNotSendError := TRUE;
	CreateMessage := TRUE;
END_IF
END_METHOD

METHOD EMStop : BOOL
VAR_INPUT
END_VAR

//nothing to do here
EMSTOP := TRUE;
END_METHOD

METHOD FB_init : BOOL
VAR_INPUT
	bInitRetains : BOOL; // if TRUE, the retain variables are initialized (warm start / cold start)
	bInCopyCode : BOOL;  // if TRUE, the instance afterwards gets moved into the copy code (online change)
END_VAR
ton_StartSMSServiceDelay(IN := TRUE);
END_METHOD

METHOD GetDiagnostics : BOOL
VAR_IN_OUT
	AddError		: ARRAY [*] OF FB_AddErrorST;
	a_ActiveEvents	: ARRAY [*] OF ST_ErrorStruct;
	w_Index			: WORD;
END_VAR
(*No emergency number configured*)	AddError[w_Index](
			b_ErrorTrig				:= get.Events.b_NoSMSNumberAvailable,
			b_SMSEnableVDL			:= FALSE,
			out_ST_Error			:= a_ActiveEvents[w_Index],
			w_ErrorID				:= 1,
			e_ObjectID				:= e_id,						//only first call set object ID.
			s_Message				:= 'no sms number available',
			e_sev					:= eSeverity.info,
			b_AutoClear				:= TRUE,
			e_ErrAckAccess			:= eErrAckAccess.General
			);
		w_Index := w_Index +1;
		
(*SMS not send warning*)	AddError[w_Index](
			b_ErrorTrig				:= get.Events.b_SMSNotSendError,
			b_SMSEnableVDL			:= FALSE,
			out_ST_Error			:= a_ActiveEvents[w_Index],
			w_ErrorID				:= 2,					
			s_Message				:= 'SMS not send',
			e_sev					:= eSeverity.info,
			b_AutoClear				:= TRUE,
			t_triggerTime			:= T#10S,
			e_ErrAckAccess			:= eErrAckAccess.General
			);
		w_Index := w_Index +1;
		
(*Modbus comm warning*)	AddError[w_Index](
			b_ErrorTrig				:= get.Events.b_MBCommWarning,
			b_SMSEnableVDL			:= FALSE,
			out_ST_Error			:= a_ActiveEvents[w_Index],
			w_ErrorID				:= 3,					
			s_Message				:= 'modbus comm. warning',
			e_sev					:= eSeverity.warning,
			b_AutoClear				:= TRUE,
			e_ErrAckAccess			:= eErrAckAccess.General
			);
		w_Index := w_Index +1;
		
(*GPS location missing*)	AddError[w_Index](
			b_ErrorTrig				:= get.Events.b_noGPSFixWarning,
			b_SMSEnableVDL			:= FALSE,
			out_ST_Error			:= a_ActiveEvents[w_Index],
			w_ErrorID				:= 5,					
			s_Message				:= 'no gps location available',
			e_sev					:= eSeverity.info,
			b_AutoClear				:= TRUE,
			e_ErrAckAccess			:= eErrAckAccess.General
			);
		w_Index := w_Index +1;
		
(*network missing*)	AddError[w_Index](
			b_ErrorTrig				:= get.Events.b_NoNetworkWarning,
			b_SMSEnableVDL			:= FALSE,
			out_ST_Error			:= a_ActiveEvents[w_Index],
			w_ErrorID				:= 6,					
			s_Message				:= 'no network available',
			e_sev					:= eSeverity.info,
			b_AutoClear				:= TRUE,
			e_ErrAckAccess			:= eErrAckAccess.General
			);
		w_Index := w_Index +1;
		
(*simcard missing*)	AddError[w_Index](
			b_ErrorTrig				:= get.Events.b_NoSimWarning,
			b_SMSEnableVDL			:= FALSE,
			out_ST_Error			:= a_ActiveEvents[w_Index],
			w_ErrorID				:= 7,					
			s_Message				:= 'no simcard available',
			e_sev					:= eSeverity.info,
			b_AutoClear				:= TRUE,
			e_ErrAckAccess			:= eErrAckAccess.General
			);
		w_Index := w_Index +1;
END_METHOD

ACTION ReadCustomRegisters:

MBRead(
	sIPAddr := st_params.IP_TELTONIKA,
	nTCPPort := st_params.MBPort_TELTONIKA,
	nUnitID := 1,
	nMBAddr := 1024,
	nQuantity := 7,//*2,
	cbLength := SIZEOF(arw_DataBuffer),
	pDestAddr := ADR(arw_DataBuffer),
	bExecute := ton_GetDataTimer.Q,
	bBusy => b_busy,
	bError => b_CommError,
	nErrId => udi_errid,
	cbRead => udi_cbread,
	tTimeout := st_params.T_MBTimeout
);

ftrig_TransmissionDone(clk := b_busy);

IF ftrig_TransmissionDone.q THEN
	IF NOT b_CommError THEN
		get.Mobile.ui_ActiveSim 		:= 	arw_DataBuffer[0];
		get.Mobile.SimStatus 			:= 	arw_DataBuffer[1];
		get.Mobile.ModemState 			:= 	arw_DataBuffer[2];
		get.Mobile.NetworkState 		:=  arw_DataBuffer[3];
		get.Wifi.WifiClienModeStatus 	:= 	arw_DataBuffer[4]; 
		get.Wifi.WifiAPModeStatus 		:= 	arw_DataBuffer[5]; 		//not yet implemented
		get.Wifi.WifiApNumberOfClients 	:= 	arw_DataBuffer[6]; 
		
			
		ui_MBRetryCount := 0;
		sfctip := TRUE;
	ELSE
		ui_MBRetryCount := ui_MBRetryCount + 1;
		sfctip := TRUE;
	END_IF
END_IF
END_ACTION

ACTION ReadDataSFC:
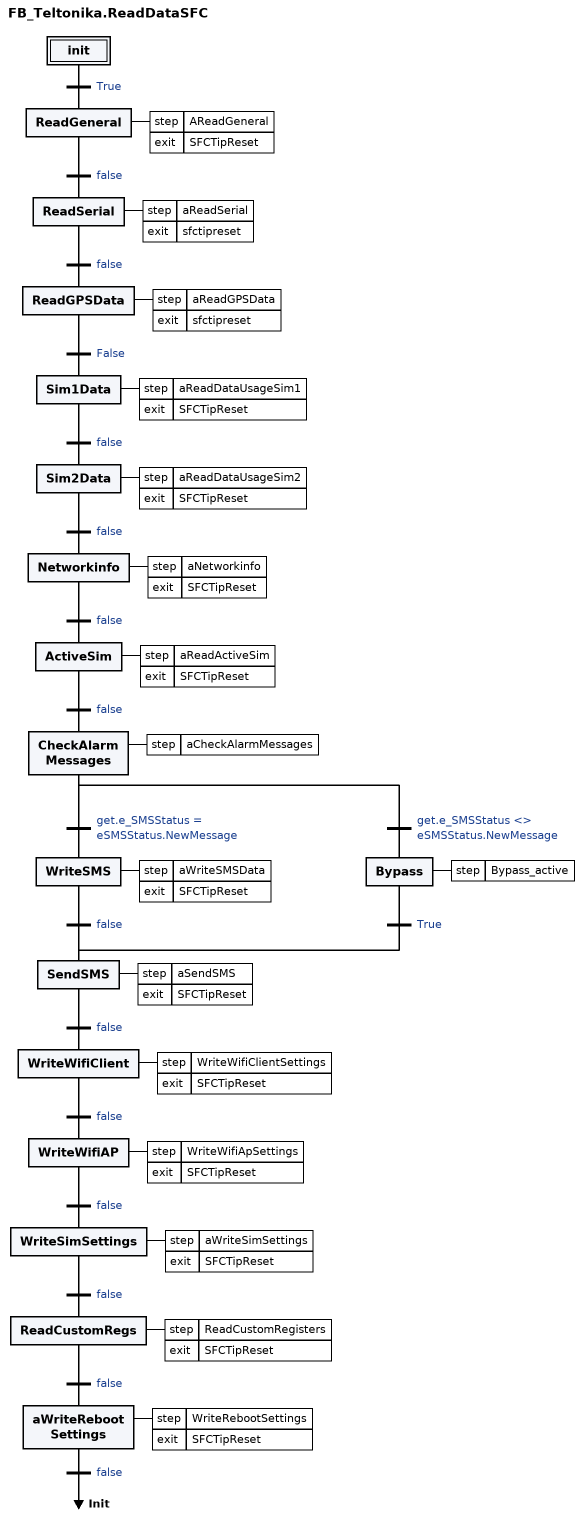
INITIAL_STEP init:
END_STEP
TRANSITION FROM init TO ReadGeneral
    := True;
END_TRANSITION
STEP ReadGeneral:
    AReadGeneral(N);  // step action
    SFCTipReset(P0);  // exit action
END_STEP
TRANSITION FROM ReadGeneral TO ReadSerial
    := false;
END_TRANSITION
STEP ReadSerial:
    aReadSerial(N);  // step action
    sfctipreset(P0);  // exit action
END_STEP
TRANSITION FROM ReadSerial TO ReadGPSData
    := false;
END_TRANSITION
STEP ReadGPSData:
    aReadGPSData(N);  // step action
    sfctipreset(P0);  // exit action
END_STEP
TRANSITION FROM ReadGPSData TO Sim1Data
    := False;
END_TRANSITION
STEP Sim1Data:
    aReadDataUsageSim1(N);  // step action
    SFCTipReset(P0);  // exit action
END_STEP
TRANSITION FROM Sim1Data TO Sim2Data
    := false;
END_TRANSITION
STEP Sim2Data:
    aReadDataUsageSim2(N);  // step action
    SFCTipReset(P0);  // exit action
END_STEP
TRANSITION FROM Sim2Data TO Networkinfo
    := false;
END_TRANSITION
STEP Networkinfo:
    aNetworkinfo(N);  // step action
    SFCTipReset(P0);  // exit action
END_STEP
TRANSITION FROM Networkinfo TO ActiveSim
    := false;
END_TRANSITION
STEP ActiveSim:
    aReadActiveSim(N);  // step action
    SFCTipReset(P0);  // exit action
END_STEP
TRANSITION FROM ActiveSim TO CheckAlarmMessages
    := false;
END_TRANSITION
STEP CheckAlarmMessages:
    aCheckAlarmMessages(N);  // step action
END_STEP
TRANSITION FROM CheckAlarmMessages TO WriteSMS
    := get.e_SMSStatus = eSMSStatus.NewMessage;
END_TRANSITION
STEP WriteSMS:
    aWriteSMSData(N);  // step action
    SFCTipReset(P0);  // exit action
END_STEP
TRANSITION FROM WriteSMS TO SendSMS
    := false;
END_TRANSITION
TRANSITION FROM CheckAlarmMessages TO Bypass
    := get.e_SMSStatus <> eSMSStatus.NewMessage;
END_TRANSITION
STEP Bypass:
    Bypass_active(N);  // step action
END_STEP
TRANSITION FROM Bypass TO SendSMS
    := True;
END_TRANSITION
STEP SendSMS:
    aSendSMS(N);  // step action
    SFCTipReset(P0);  // exit action
END_STEP
TRANSITION FROM SendSMS TO WriteWifiClient
    := false;
END_TRANSITION
STEP WriteWifiClient:
    WriteWifiClientSettings(N);  // step action
    SFCTipReset(P0);  // exit action
END_STEP
TRANSITION FROM WriteWifiClient TO WriteWifiAP
    := false;
END_TRANSITION
STEP WriteWifiAP:
    WriteWifiApSettings(N);  // step action
    SFCTipReset(P0);  // exit action
END_STEP
TRANSITION FROM WriteWifiAP TO WriteSimSettings
    := false;
END_TRANSITION
STEP WriteSimSettings:
    aWriteSimSettings(N);  // step action
    SFCTipReset(P0);  // exit action
END_STEP
TRANSITION FROM WriteSimSettings TO ReadCustomRegs
    := false;
END_TRANSITION
STEP ReadCustomRegs:
    ReadCustomRegisters(N);  // step action
    SFCTipReset(P0);  // exit action
END_STEP
TRANSITION FROM ReadCustomRegs TO aWriteRebootSettings
    := false;
END_TRANSITION
STEP aWriteRebootSettings:
    WriteRebootSettings(N);  // step action
    SFCTipReset(P0);  // exit action
END_STEP
TRANSITION FROM aWriteRebootSettings TO Init
    := false;
END_TRANSITION
// branch label Branch0_ReadDataSFC
END_ACTION

METHOD Reset : BOOL
VAR_INPUT
END_VAR
get.Events.b_SMSNotSendError := FALSE;
get.e_SMSStatus := eSMSStatus.Idle;

Reset := TRUE;
END_METHOD

METHOD SetDevName : BOOL
VAR_INPUT
	s_DevName	:	String(12);
END_VAR
IF s_DevName = '' THEN
	get.Mobile.s_EmergencySMSDevName := ''; //<-- stParams.serial number
ELSE
	get.Mobile.s_EmergencySMSDevName :=	s_DevName;
END_IF

SetDevName := get.Mobile.s_EmergencySMSDevName <> '';
END_METHOD

METHOD SetSMSNumber : BOOL
VAR_INPUT
	s_SMSNumber	:	STRING(20);
END_VAR
VAR 
	for_counter	:	UINT :=0;
	InternalString	:	STRING(20);
	intermediateValue	:	UINT;
	
	temp	:	string(10);
END_VAR

SetSMSNumber := TRUE;

//check minimum length
IF INT_TO_UINT(len(s_SMSNumber)) < st_params.MinimumPhoneNumberLength AND s_SMSNumber <> '' THEN
	SetSMSNumber := FALSE;
ELSE
	InternalString := s_SMSNumber;
	
	//replace leading + with 00
	IF left(InternalString,1) = '+' THEN
		InternalString := Replace(InternalString, '00', 1, 1);
	END_IF
	
	//check for non_numeric characters
	FOR for_counter := 1 TO INT_TO_UINT(len(InternalString)) DO
		intermediateValue := f_toASC(mid(InternalString, 1, UINT_TO_INT(for_counter)));
		IF (intermediateValue < 48 OR intermediateValue > 57) THEN
			SetSMSNumber := FALSE;
		END_IF
	END_FOR
END_IF

//only if all checks succeed, the number is written to the struct.
IF SetSMSNumber THEN
	get.Mobile.s_EmergencySMSNumber := InternalString;
ELSE
	get.Mobile.s_EmergencySMSNumber := '';
END_IF

get.Events.b_NoSMSNumberAvailable := NOT SetSMSNumber;
END_METHOD

ACTION SFCTipReset:
SFCTip := FALSE;
END_ACTION

ACTION WriteRebootSettings:

arw_DataBuffer[0] := TO_UINT(set.AutoRebootEnable);
arw_DataBuffer[1] := TO_UINT(set.ManualReboot);

MBWrite(
	sIPAddr := st_params.IP_TELTONIKA,
	nTCPPort := st_params.MBPort_TELTONIKA,
	nUnitID := 1,
	nMBAddr := 1139,
	nQuantity := 2,
	cbLength := SIZEOF(arw_DataBuffer),
	pSrcAddr	:=	ADR(arw_DataBuffer),
	bExecute := ton_GetDataTimer.Q,
	bBusy => b_busy,
	bError => b_CommError,
	nErrId => udi_errid,
	tTimeout := st_params.T_MBTimeout
);

ftrig_TransmissionDone(clk := b_busy);

IF ftrig_TransmissionDone.q THEN
	sfctip := TRUE;
	set.ManualReboot := false;
END_IF
END_ACTION

ACTION WriteWifiAPSettings:

arw_DataBuffer[0] := TO_UINT(set.EnableWifiAP);
memcpy(ADR(arw_DataBuffer[1]), ADR(set.WifiAPSSID), 32);
memcpy(ADR(arw_DataBuffer[17]), ADR(set.WifiAPPass), 32);
arw_DataBuffer[33] := TO_UINT(set.WifiAPSecType);

FOR ui_counter := 1 TO 32 DO
	arw_DataBuffer[ui_counter] := host_to_be16(arw_DataBuffer[ui_counter]);
END_FOR

MBWrite(
	sIPAddr := st_params.IP_TELTONIKA,
	nTCPPort := st_params.MBPort_TELTONIKA,
	nUnitID := 1,
	nMBAddr := 1099,
	nQuantity := 34,
	cbLength := SIZEOF(arw_DataBuffer),
	pSrcAddr	:=	ADR(arw_DataBuffer),
	bExecute := ton_GetDataTimer.Q,
	bBusy => b_busy,
	bError => b_CommError,
	nErrId => udi_errid,
	tTimeout := st_params.T_MBTimeout
);

ftrig_TransmissionDone(clk := b_busy);

IF ftrig_TransmissionDone.q THEN
		sfctip := TRUE;
END_IF
END_ACTION

ACTION WriteWifiClientSettings:

arw_DataBuffer[0] := TO_UINT(set.EnableWifiClient);
memcpy(ADR(arw_DataBuffer[1]), ADR(set.WifiClientSSID), 32);
memcpy(ADR(arw_DataBuffer[17]), ADR(set.WifiClientPass), 32);
arw_DataBuffer[33] := TO_UINT(set.WifiClientSecType);

FOR ui_counter := 1 TO 32 DO
	arw_DataBuffer[ui_counter] := host_to_be16(arw_DataBuffer[ui_counter]);
END_FOR

MBWrite(
	sIPAddr := st_params.IP_TELTONIKA,
	nTCPPort := st_params.MBPort_TELTONIKA,
	nUnitID := 1,
	nMBAddr := 1059,
	nQuantity := 34,
	cbLength := SIZEOF(arw_DataBuffer),
	pSrcAddr	:=	ADR(arw_DataBuffer),
	bExecute := ton_GetDataTimer.Q,
	bBusy => b_busy,
	bError => b_CommError,
	nErrId => udi_errid,
	tTimeout := st_params.T_MBTimeout
);

ftrig_TransmissionDone(clk := b_busy);

IF ftrig_TransmissionDone.q THEN
		sfctip := TRUE;
END_IF
END_ACTION

END_FUNCTION_BLOCK

// ---- POUs/ErrorHandling/FB_AddErrorST.TcPOU
FUNCTION_BLOCK FB_AddErrorST
VAR PERSISTENT
	b_SMSenableUser				: BOOL;
END_VAR

VAR_INPUT
	b_ErrorTrig					: BOOL;
	b_SMSEnableVDL				: BOOL;
	t_TriggerTime				: TIME := T#0S;
	b_AutoClear					: BOOL := FALSE;
	e_ErrAckAccess				: eErrAckAccess := eErrAckAccess.VDL; //default full access required
	w_ErrorID					: WORD;
	e_objectID					: eObject_ID :=  eObject_ID.None;
	s_message					: STRING;
	e_sev						: eSeverity;
END_VAR
VAR_IN_OUT
	out_st_Error 				: ST_ErrorStruct;
END_VAR

VAR_OUTPUT
	b_out						: BOOL;
END_VAR

VAR
	i_instance					: INT;
	b_clear						: BOOL;
	s_MessageOld				: STRING;
	b_MessageChanged			: BOOL;
	b_SetError					: BOOL;
	sr_ErrorActive				: SR;
	bIsInitialized 				: BOOL := FALSE;	
	ton_FaultTriggerTime		: TON;
	fTRIG_Fault					: F_TRIG;
	rTRIG_Fault					: R_TRIG;
	
	b_clearCommand				: BOOL;
	
	//FOR SMS MESSAGE FUNCTIONALITY
	b_SetSMSmessage				: BOOL;
	b_ClearSMSmessage			: BOOL;
	s_SMSmessage				: STRING;
	i_SMSMessageIndex			: INT;
END_VAR

VAR_STAT
	i_instanceCounter			: INT;
	e_objectID_static			: eObject_ID;
END_VAR

//set object ID if given and not same as it was.
IF e_objectID <> 0 AND e_objectID <> e_objectID_static THEN 
	e_objectID_static := e_objectID;
END_IF

IF NOT bIsInitialized THEN
	//SET default SMS enable	
	out_st_error.b_SMSEnable := b_SMSEnableVDL OR b_SMSenableUser;
	//SET error ID
	out_st_Error.w_ID		:= w_ErrorID + e_objectID_static;
	//SET severity
	out_st_Error.s_Severity	:= TO_STRING(e_Sev);
	//SET instance
	IF w_ErrorID <> 0 THEN
		i_instanceCounter := i_instanceCounter +1;
	END_IF
	i_instance := i_instanceCounter;
	
	bIsInitialized := TRUE;		
ELSE
	//only allow user setting when vdl default is not set.
	IF NOT b_SMSEnableVDL AND b_SMSenableUser <> out_st_error.b_SMSEnable THEN
		b_SMSenableUser := out_st_error.b_SMSEnable;
	END_IF
END_IF

b_MessageChanged := s_MessageOld <> s_Message;
IF b_MessageChanged THEN
	// set last stored value
	s_MessageOld := s_Message;
	// The code that you want to be executed at the first cycle or on change
	out_st_Error.s_Message	:= Concat(Concat(TO_STRING(e_objectID_static),' - '), s_message);
	s_SMSmessage := CONCAT(CONCAT(out_st_Error.s_Severity, ': '), out_st_Error.s_Message);
END_IF

ton_FaultTriggerTime(IN:= b_ErrorTrig, PT:= t_TriggerTime);
b_out := ton_FaultTriggerTime.Q;
out_st_error.b_ErrorActive := b_out;


IF b_out THEN	
	//Also write diagnostics to SystemLog
	CASE e_sev OF
		eSeverity.Warning 			: GVL.b_WarningActive := TRUE;
		eSeverity.Normalshutdown 	: GVL.b_NormalshutdownActive := TRUE;
		eSeverity.Quickshutdown 	: GVL.b_QuickShutdownActive := TRUE;
		eSeverity.EmergencyShutdown	: GVL.b_EmergencyShutdownActive := TRUE;
	END_CASE
END_IF

rTRIG_Fault(CLK := b_Out);
b_SetError := rTRIG_Fault.Q OR (out_st_Error.s_DateError = '' AND b_out);
IF b_SetError AND GVL.b_SystemClockOK THEN;
	//WriteLogItem(Source := e_objectID, Severity := e_sev, LogText := s_message);
	out_st_Error.s_DateError := GVL.s_SystemDate;
	out_st_Error.s_TimeError := GVL.s_SystemTime;
	out_st_Error.s_TimeCleared	:= '';
	
	//for sms service
	b_SetSMSmessage := TRUE;
END_IF

//CLEARING
b_Clear := b_AutoClear AND e_Sev < eSeverity.NormalShutdown AND NOT b_ErrorTrig;
IF (ErrorHandling.tp_Clearevents.Q OR b_Clear) AND out_st_Error.s_TimeCleared <> '' THEN
	b_ClearCommand := TRUE;
END_IF

//CLEARING EVENTS
IF b_ClearCommand THEN
	out_st_Error.s_DateError 	:= '';
	out_st_Error.s_TimeError 	:= '';
	out_st_Error.s_TimeCleared	:= '';
	b_ClearCommand := FALSE;
END_IF

fTRIG_Fault(CLK := b_Out);
IF out_st_Error.s_TimeError <> '' AND fTRIG_Fault.Q THEN;
	out_st_Error.s_TimeCleared	:= GVL.s_SystemTime;
	b_ClearSMSmessage := TRUE;
END_IF

///SMS message buffer
IF b_SetSMSmessage AND (b_SMSEnableVDL OR b_SMSenableUser) THEN
	IF AppendMessage(
		as_buffer := errorhandling.a_SMSEventBuffer, 
		s_message := s_SMSmessage, 
		index=> i_SMSMessageIndex) THEN
		 	b_SetSMSmessage := FALSE;
	END_IF 
ELSIF b_clearSMSmessage THEN
	IF DeleteMessage(as_buffer := errorhandling.a_SMSEventBuffer, index := i_SMSMessageIndex ) THEN
		b_ClearSMSmessage := FALSE;
	END_IF
END_IF

METHOD AppendMessage : BOOL;
VAR_IN_OUT
	as_buffer	: ARRAY [*] OF STRING;
END_VAR

VAR_INPUT
	s_message : STRING;
END_VAR
VAR_OUTPUT
	index : INT;
END_VAR

VAR
	i: INT;
END_VAR
AppendMessage := FALSE;

FOR i:= TO_INT(LOWER_BOUND(as_buffer,1)) TO TO_INT(UPPER_BOUND(as_buffer,1)) DO
	IF as_buffer[i] = '' THEN
		as_buffer[i] := s_message;
		index := i;
		AppendMessage := TRUE;
		EXIT;
	END_IF	
END_FOR
END_METHOD

METHOD DeleteMessage : BOOL

VAR_IN_OUT
	as_buffer	: ARRAY [*] OF STRING;
END_VAR

VAR_INPUT
	index		: INT;
END_VAR
DeleteMessage := FALSE;
as_buffer[index] := '';

IF as_buffer[index] = '' THEN
	DeleteMessage := TRUE;
END_IF
END_METHOD

END_FUNCTION_BLOCK

// ---- POUs/ErrorHandling/ErrorHandling.TcPOU
PROGRAM INTERNAL ErrorHandling
VAR_INPUT
	e_access					: eErrAckAccess;
	b_ClearEvents				: BOOL;	
	AddError					: ARRAY [0..i_maxevents] OF FB_addErrorST;
END_VAR

VAR	
	tp_ClearEvents						: TP := (PT := T#1S);
	a_SMSEventBuffer					: ARRAY [1..10] OF STRING;
	ton_ErrorMessageOnDelay				: TON := (PT:= T#10S);
	
	//Errorhandling
	w_ErrorIndex				: WORD;
	w_Totalerrors				: WORD;
	b_ResetError				: BOOL;
	(*ENUM*)
	
	//Refresh Timer
	ton_RefreshTimer						: TON := (PT:= T#500MS);
	b_refreshErrors							: BOOL;
	b_initCycle								: BOOL := TRUE;
	{ attribute 'TcHmiSymbol.ShowRecursively'}
	a_ActiveEvents							: ARRAY [0..i_maxevents	] OF ST_ErrorStruct;
	
	
	r_trigNormalShutdown					: R_TRIG;
END_VAR

VAR_OUTPUT
	w_errorword							: WORD;
	b_QuickShutdownActive				: BOOL;
	b_NormalShutdownTrigger				: BOOL;
END_VAR

VAR CONSTANT
	i_maxevents							: INT := 400;
END_VAR

//Reset variables
w_ErrorIndex 					:= 0;

//RealtimeClock
SystemClock();

//clear pulse
tp_ClearEvents(IN := b_ClearEvents);

//ONdelay
ton_ErrorMessageOnDelay(IN:= NOT b_InitCycle);

//Refresh signal
ton_RefreshTimer(IN:= NOT(ton_RefreshTimer.Q));
b_RefreshErrors := ton_RefreshTimer.Q OR b_InitCycle;
IF b_RefreshErrors AND ton_ErrorMessageOnDelay.Q THEN
	GVL.b_WarningActive				:= FALSE;
	GVL.b_NormalShutdownActive		:= FALSE;
	GVL.b_QuickshutdownActive		:= FALSE;
	GVL.b_EmergencyShutdownActive	:= FALSE;	

	Safety.GetDiagnostics(AddError, a_ActiveEvents, w_errorindex);
	Main_Fast.PowerMonitor.GetDiagnostics(AddError, a_ActiveEvents,  w_errorindex);
	Main_Fast.InternalPowerSupply.GetDiagnostics(AddError, a_ActiveEvents, w_errorindex);
	Main_Fast.NeutralTransformer.GetDiagnostics(AddError, a_ActiveEvents, w_errorindex);
	Main_Fast.HartingIO.GetDiagnostics(AddError, a_ActiveEvents, w_errorindex);
	Main_Fast.PowerStack.GetDiagnostics(AddError, a_ActiveEvents, w_errorindex);
	Main_Fast.Protectionsystems.GetDiagnostics(AddError, a_ActiveEvents, w_errorindex);
	Main_Fast.BMS.GetDiagnostics(AddError, a_ActiveEvents, w_errorindex);
	Main_Fast.Enclosure.GetDiagnostics(AddError, a_ActiveEvents, w_errorindex);
	Main_Fast.Coolingsystem.GetDiagnostics(AddError, a_ActiveEvents, w_errorindex);
	Main_Fast.ACswitchgear.GetDiagnostics(AddError, a_ActiveEvents, w_errorindex);
	Main_Fast.Router.GetDiagnostics(AddError, a_ActiveEvents, w_errorindex);
	controlmanager.PNController.GetDiagnostics(AddError, a_ActiveEvents, w_errorindex);
	Main_Fast.SystemControl.GetDiagnostics(AddError, a_ActiveEvents, w_errorindex);
	Main_Fast.Peakshavebox.GetDiagnostics(AddError, a_ActiveEvents, w_errorindex);
	Main_Fast.GenComm.GetDiagnostics(AddError, a_ActiveEvents, w_errorindex);
	Main_Fast.AcDcCharger.GetDiagnostics(AddError, a_ActiveEvents, w_errorindex);
	controlmanager.IoT.GetDiagnostics(AddError, a_ActiveEvents, w_errorindex);
	w_Totalerrors := w_errorindex;
END_IF

//If larger than 0, error is existing
b_QuickShutdownActive := GVL.b_QuickshutdownActive OR GVL.b_EmergencyShutdownActive;
r_trigNormalShutdown(CLK := GVL.b_NormalShutdownActive, Q => b_normalShutdownTrigger);

b_initCycle := FALSE;

END_PROGRAM

// ---- POUs/Functions-FBs-Programs/_PRGS/SystemClock.TcPOU
PROGRAM SystemClock
VAR
	ton_RefreshTime			: TON :=(PT:= T#10mS);
	fb_GetLocalSystemtime 	: FB_localSystemTime;
	s_systemDateTime		: STRING(40);
END_VAR

ton_RefreshTime(IN:= NOT(ton_RefreshTime.Q));

IF ton_RefreshTime.Q THEN
	fb_GetLocalSystemtime(
		bEnable := TRUE,
		dwCycle := 1);
	s_SystemDateTime := SYSTEMTIME_TO_STRING(fb_GetLocalSystemtime.systemTime);
	gvl.dt_SystemDateTime := SYSTEMTIME_TO_DT(fb_GetLocalSystemtime.systemTime);
	GVL.s_SystemDate := MID(s_SystemDateTime, 10, 1);
	GVL.s_SystemTime := MID(s_SystemDateTime, 12, 12);
END_IF

GVL.b_SystemClockOK := GVL.s_SystemDate <> '1970-01-01' AND GVL.s_SystemTime <> '00:00:00';

END_PROGRAM

// ---- POUs/Safety/Safety.TcPOU
PROGRAM Safety
	{attribute 'TcContextId':='0'}
VAR
	ToSafetyPrg							AT %Q* : ST_Safety_ToSafetyPrg;
	b_ManualReset								: BOOL;
	
	ton_Reset									: Ton := (PT:=T#100MS);
	
	PowerModuleDoorSwitch	:	FB_VarLogger;
	EMstopSwitch			:	FB_VarLogger;	
	SafetyStopCount			:	FB_VarLogger;
END_VAR

VAR_INPUT
	EDMSignals								: ST_Safety_ContactorEDM;
	b_enable									: BOOL;
	b_extEmstopTrigger						: BOOL;
END_VAR

VAR_OUTPUT
	// FROM Safety (feedbacks)
	get									AT %I* : ST_Safety_get;	
END_VAR

IF NOT b_enable OR b_manualReset THEN
	ToSafetyPrg.b_safetyPRGReset := TRUE;
	ToSafetyPrg.b_ErrorReset := TRUE;
ELSE
	ToSafetyPrg.b_safetyPRGReset := FALSE;
	ToSafetyPrg.b_ErrorReset := FALSE;
END_IF

//Couple EDM signals
ToSafetyPrg.contactors.b_NetcontactorEDM := EDMSignals.b_NetcontactorEDM;
ToSafetyPrg.contactors.b_MccbMasterEDM := EDMSignals.b_MccbMasterEDM;
ToSafetyPrg.contactors.b_MccbSlaveEDM := EDMSignals.b_MccbSlaveEDM;

// SEND software E-stop to safety prg,so when quickshutdown is given from normal program, safety shutsdown. Also HMI e-stop can activate software e-stop.
ToSafetyPrg.b_emergencyStopSoftwareOK := NOT(GVL.b_QuickshutdownActive OR b_extEmstopTrigger);

ton_Reset();

METHOD PUBLIC GetDiagnostics
VAR_IN_OUT
	AddError		: ARRAY [*] OF FB_AddErrorST;
	a_ActiveEvents	: ARRAY [*] OF ST_ErrorStruct;
	w_Index			: WORD;
END_VAR
(*EmergencyStop ChA*)		AddError[w_Index](
		b_ErrorTrig			:= NOT(get.b_EStopChannelAOK),
		out_ST_Error			:= a_ActiveEvents[w_Index],
		w_ErrorID					:= 1,
		e_ObjectID				:= eObject_ID.Safety,
		s_Message				:= 'channel A',
		b_SMSEnableVDL			:= TRUE,
		e_sev					:= eseverity.EmergencyShutdown,
	);
	w_Index := w_Index +1;
	
	(*EmergencyStop ChB*)		AddError[w_Index](
		b_ErrorTrig			:= NOT(get.b_EStopChannelBOK),
		out_ST_Error			:= a_ActiveEvents[w_Index],
		w_ErrorID					:= 2,
		s_Message				:= 'channel B',
		e_sev					:= eseverity.EmergencyShutdown,
	);
	w_Index := w_Index +1;
	
	(*EmergencyStop MRCDB*)		AddError[w_Index](
		b_ErrorTrig			:= NOT(get.b_MRCDBOK),
		out_ST_Error			:= a_ActiveEvents[w_Index],
		w_ErrorID					:= 3,
		s_Message				:= 'residual current fault detected',
		e_sev					:= eseverity.EmergencyShutdown,
		b_SMSEnableVDL		:= TRUE,
	);
	w_Index := w_Index +1;
	
	(*EmergencyStop Insulation*)AddError[w_Index](
		b_ErrorTrig			:= NOT(get.b_InsulationMonitorOK),
		out_ST_Error			:= a_ActiveEvents[w_Index],
		w_ErrorID					:= 4,
		s_Message				:= 'insulation fault detected',
		e_sev					:= eseverity.EmergencyShutdown,
		b_SMSEnableVDL		:= TRUE,
	);
	w_Index := w_Index +1;
	
	(*EmergencyStop Inverter Door*) AddError[w_Index](
		b_ErrorTrig			:= NOT(get.b_InverterDoorOK),
		out_ST_Error			:= a_ActiveEvents[w_Index],
		w_ErrorID					:= 5,
		s_Message				:= 'inverter door opened',
		e_sev					:= eseverity.EmergencyShutdown,
		b_SMSEnableVDL		:= TRUE,
	);
	w_Index := w_Index +1;
	
	(*EmergencyStop ZPT-OCP *) AddError[w_Index](
		b_ErrorTrig			:= NOT(get.b_ZptOK),
		out_ST_Error			:= a_ActiveEvents[w_Index],
		w_ErrorID					:= 6,
		s_Message				:= 'ZPT overcurrent trip',
		e_sev					:= eseverity.EmergencyShutdown,
		b_SMSEnableVDL		:= TRUE,
	);
	w_Index := w_Index +1;
	
(*EmergencyStop initiated*) AddError[w_Index](
		b_ErrorTrig			:= NOT(get.b_SafetyOK),
		out_ST_Error			:= a_ActiveEvents[w_Index],
		w_ErrorID					:= 10,
		s_Message				:= 'emergency stop initiated',
		e_sev					:= eseverity.EmergencyShutdown,
		b_SMSEnableVDL		:= FALSE,
	);
	w_Index := w_Index +1;
END_METHOD

METHOD GetWearCounters : BOOL
VAR_INPUT
END_VAR
PowerModuleDoorSwitch(	TriggerInput := NOT get.b_InverterDoorOK, 
						LogItemGroup :=  eLogItemGroupID.Safety, 
						LogItemName := 'InvDoorSwCnt', 
						LogType := eLogTypes.TrackCycles);

